SPLINE
SPL {X  -165.650, Y  +635.985, Z    +0.000, E1   -68.274, E3 +149186.290}
SPL {X  -165.650, Y  +656.072, Z    +0.000, E1   -68.403, E3 +149201.585}
SPL {X  -165.650, Y  +673.246, Z    +0.000, E1   -68.189, E3 +149217.340}
SPL {X  -164.760, Y  +692.647, Z    +0.000, E1   -68.400, E3 +149231.305}
SPL {X  -162.986, Y  +705.089, Z    +0.000, E1   -67.915, E3 +149245.517}
SPL {X  -160.378, Y  +716.957, Z    +0.000, E1   -67.874, E3 +149255.337}
SPL {X  -157.774, Y  +725.970, Z    +0.000, E1   -67.383, E3 +149266.685}
SPL {X  -154.751, Y  +734.593, Z    +0.000, E1   -66.864, E3 +149277.279}
SPL {X  -151.443, Y  +742.618, Z    +0.000, E1   -66.527, E3 +149286.274}
SPL {X  -148.198, Y  +749.508, Z    +0.000, E1   -66.065, E3 +149294.755}
SPL {X  -144.642, Y  +756.238, Z    +0.000, E1   -65.678, E3 +149302.621}
SPL {X  -140.398, Y  +763.411, Z    +0.000, E1   -64.853, E3 +149313.097}
SPL {X  -135.180, Y  +771.240, Z    +0.000, E1   -64.104, E3 +149323.147}
SPL {X  -125.028, Y  +784.164, Z    +0.000, E1   -66.760, E3 +149321.617}
SPL {X   -71.589, Y  +824.882, Z    +0.000, E1   -56.415, E3 +149448.682}
ENDSPLINE

SPLINE
SPL {X  -127.072, Y  +781.767, Z    +0.000, E1   -54.186, E3 +149611.654}
SPL {X  -150.680, Y  +744.314, Z    +0.000, E1   -44.608, E3 +149622.610}
SPL {X  -160.361, Y  +717.026, Z    +0.000, E1   -30.396, E3 +149611.464}
SPL {X  -163.361, Y  +702.946, Z    +0.000, E1   -22.646, E3 +149616.583}
SPL {X  -165.092, Y  +689.091, Z    +0.000, E1   -12.938, E3 +149616.153}
SPL {X  -165.629, Y  +678.122, Z    +0.000, E1    -4.178, E3 +149615.300}
SPL {X  -165.650, Y  +673.290, Z    +0.000, E1    +0.167, E3 +149614.256}
SPL {X  -165.650, Y  +669.039, Z    +0.000, E1    +7.218, E3 +149613.603}
SPL {X  -165.650, Y  +663.739, Z    +0.000, E1   +17.756, E3 +149613.294}
SPL {X  -165.650, Y  +659.573, Z    +0.000, E1   +26.182, E3 +149613.147}
SPL {X  -165.650, Y  +652.464, Z    +0.000, E1   +39.379, E3 +149612.188}
SPL {X  -165.650, Y  +634.871, Z    +0.000, E1   +61.762, E3 +149609.421}
SPL {X  -165.650, Y  +574.769, Z    +0.000, E1   +74.441, E3 +149622.069}
SPL {X  -165.650, Y  +420.321, Z    +0.000, E1   +71.570, E3 +149713.074}
ENDSPLINE

SPLINE
SPL {X  -165.650, Y  +437.633, Z    +0.000, E1   +68.421, E3 +149728.822}
ENDSPLINE

SPLINE
SPL {X  -164.513, Y  +359.128, Z    +0.000, E1   +73.170, E3 +149739.056}
SPL {X  -163.967, Y  +354.944, Z    +0.000, E1   +72.327, E3 +149750.409}
SPL {X  -163.372, Y  +351.124, Z    +0.000, E1   +71.295, E3 +149763.001}
SPL {X  -162.653, Y  +347.134, Z    +0.000, E1   +70.371, E3 +149774.237}
SPL {X  -161.430, Y  +341.349, Z    +0.000, E1   +69.492, E3 +149786.311}
SPL {X  -160.389, Y  +337.084, Z    +0.000, E1   +68.301, E3 +149799.398}
SPL {X  -159.245, Y  +332.881, Z    +0.000, E1   +67.496, E3 +149809.058}
SPL {X  -157.072, Y  +325.885, Z    +0.000, E1   +67.020, E3 +149818.407}
SPL {X  -154.432, Y  +318.577, Z    +0.000, E1   +66.843, E3 +149825.612}
SPL {X  -151.047, Y  +310.495, Z    +0.000, E1   +66.593, E3 +149834.024}
SPL {X  -146.639, Y  +301.448, Z    +0.000, E1   +65.839, E3 +149846.233}
SPL {X  -142.469, Y  +293.987, Z    +0.000, E1   +65.133, E3 +149856.282}
SPL {X  -139.022, Y  +288.429, Z    +0.000, E1   +64.807, E3 +149862.480}
SPL {X  -136.717, Y  +284.968, Z    +0.000, E1   +64.044, E3 +149869.073}
SPL {X  -133.061, Y  +279.835, Z    +0.000, E1   +64.204, E3 +149872.486}
SPL {X  -118.927, Y  +263.191, Z    +0.000, E1   +67.951, E3 +149868.499}
SPL {X   -76.819, Y  +231.739, Z    +0.000, E1   +54.834, E3 +150046.505}
ENDSPLINE

SPLINE
SPL {X  -140.879, Y  +291.363, Z    +0.000, E1   +48.273, E3 +150153.946}
SPL {X  -158.845, Y  +331.507, Z    +0.000, E1   +33.834, E3 +150163.281}
SPL {X  -164.164, Y  +356.358, Z    +0.000, E1   +18.707, E3 +150159.604}
SPL {X  -165.341, Y  +368.384, Z    +0.000, E1   +10.076, E3 +150160.348}
SPL {X  -165.648, Y  +377.641, Z    +0.000, E1    +2.653, E3 +150159.698}
SPL {X  -165.650, Y  +380.939, Z    +0.000, E1    -0.407, E3 +150158.509}
SPL {X  -165.650, Y  +385.900, Z    +0.000, E1    -8.711, E3 +150157.954}
SPL {X  -165.650, Y  +390.854, Z    +0.000, E1   -18.692, E3 +150157.129}
SPL {X  -165.650, Y  +395.801, Z    +0.000, E1   -28.236, E3 +150157.128}
SPL {X  -165.650, Y  +403.802, Z    +0.000, E1   -41.748, E3 +150156.949}
SPL {X  -165.650, Y  +418.088, Z    +0.000, E1   -59.974, E3 +150154.222}
SPL {X  -165.650, Y  +461.994, Z    +0.000, E1   -72.657, E3 +150162.360}
SPL {X  -165.650, Y  +492.072, Z    +0.000, E1   -73.925, E3 +150172.462}
SPL {X  -165.650, Y  +640.142, Z    +0.000, E1   -72.635, E3 +150251.338}
ENDSPLINE

SPLINE
SPL {X  -165.650, Y  +612.217, Z    +0.000, E1   -68.647, E3 +150267.263}
ENDSPLINE

SPLINE
SPL {X  -165.650, Y  +623.643, Z    +0.000, E1   -68.543, E3 +150277.360}
SPL {X  -165.650, Y  +635.985, Z    +0.000, E1   -68.274, E3 +150289.739}
SPL {X  -165.650, Y  +647.687, Z    +0.000, E1   -68.151, E3 +150300.238}
SPL {X  -165.650, Y  +665.917, Z    +0.000, E1   -68.414, E3 +150312.998}
SPL {X  -165.417, Y  +684.287, Z    +0.000, E1   -68.467, E3 +150327.295}
SPL {X  -164.655, Y  +693.631, Z    +0.000, E1   -68.130, E3 +150337.646}
SPL {X  -162.986, Y  +705.089, Z    +0.000, E1   -67.915, E3 +150348.965}
SPL {X  -159.812, Y  +719.091, Z    +0.000, E1   -67.711, E3 +150361.964}
SPL {X  -156.969, Y  +728.420, Z    +0.000, E1   -67.278, E3 +150372.746}
SPL {X  -154.751, Y  +734.593, Z    +0.000, E1   -66.864, E3 +150380.727}
SPL {X  -151.443, Y  +742.618, Z    +0.000, E1   -66.527, E3 +150389.722}
SPL {X  -148.198, Y  +749.508, Z    +0.000, E1   -66.065, E3 +150398.203}
SPL {X  -144.642, Y  +756.238, Z    +0.000, E1   -65.678, E3 +150406.070}
SPL {X  -140.398, Y  +763.411, Z    +0.000, E1   -64.853, E3 +150416.546}
SPL {X  -135.180, Y  +771.240, Z    +0.000, E1   -64.104, E3 +150426.595}
SPL {X  -125.028, Y  +784.164, Z    +0.000, E1   -66.760, E3 +150425.065}
SPL {X   -71.589, Y  +824.882, Z    +0.000, E1   -56.415, E3 +150552.130}
ENDSPLINE

SPLINE
SPL {X  -127.072, Y  +781.767, Z    +0.000, E1   -54.186, E3 +150715.102}
SPL {X  -150.680, Y  +744.314, Z    +0.000, E1   -44.608, E3 +150726.059}
SPL {X  -162.376, Y  +708.273, Z    +0.000, E1   -25.870, E3 +150718.182}
SPL {X  -165.092, Y  +689.091, Z    +0.000, E1   -12.938, E3 +150719.601}
SPL {X  -165.629, Y  +678.122, Z    +0.000, E1    -4.178, E3 +150718.748}
SPL {X  -165.650, Y  +673.539, Z    +0.000, E1    -0.057, E3 +150717.846}
SPL {X  -165.650, Y  +671.359, Z    +0.000, E1    +3.116, E3 +150717.203}
SPL {X  -165.650, Y  +667.465, Z    +0.000, E1   +10.413, E3 +150716.997}
SPL {X  -165.650, Y  +662.220, Z    +0.000, E1   +20.600, E3 +150716.689}
SPL {X  -165.650, Y  +652.464, Z    +0.000, E1   +39.379, E3 +150715.637}
SPL {X  -165.650, Y  +636.657, Z    +0.000, E1   +60.410, E3 +150712.925}
SPL {X  -165.650, Y  +613.310, Z    +0.000, E1   +72.038, E3 +150713.284}
SPL {X  -165.650, Y  +568.914, Z    +0.000, E1   +74.438, E3 +150727.869}
SPL {X  -165.650, Y  +420.321, Z    +0.000, E1   +71.570, E3 +150816.522}
ENDSPLINE

SPLINE
SPL {X  -165.650, Y  +437.633, Z    +0.000, E1   +68.421, E3 +150832.270}
ENDSPLINE

SPLINE
SPL {X  -164.513, Y  +359.128, Z    +0.000, E1   +73.170, E3 +150842.504}
SPL {X  -163.967, Y  +354.944, Z    +0.000, E1   +72.327, E3 +150853.857}
SPL {X  -163.372, Y  +351.124, Z    +0.000, E1   +71.295, E3 +150866.450}
SPL {X  -162.653, Y  +347.134, Z    +0.000, E1   +70.371, E3 +150877.685}
SPL {X  -161.451, Y  +341.438, Z    +0.000, E1   +69.889, E3 +150886.004}
SPL {X  -161.195, Y  +340.340, Z    +0.000, E1   +68.690, E3 +150897.225}
SPL {X  -159.328, Y  +333.173, Z    +0.000, E1   +67.752, E3 +150910.445}
SPL {X  -157.072, Y  +325.885, Z    +0.000, E1   +67.020, E3 +150921.855}
SPL {X  -154.432, Y  +318.577, Z    +0.000, E1   +66.843, E3 +150929.060}
SPL {X  -151.047, Y  +310.495, Z    +0.000, E1   +66.593, E3 +150937.472}
SPL {X  -146.639, Y  +301.448, Z    +0.000, E1   +65.839, E3 +150949.682}
SPL {X  -142.469, Y  +293.987, Z    +0.000, E1   +65.133, E3 +150959.730}
SPL {X  -139.022, Y  +288.429, Z    +0.000, E1   +64.807, E3 +150965.929}
SPL {X  -136.717, Y  +284.968, Z    +0.000, E1   +64.044, E3 +150972.521}
SPL {X  -133.061, Y  +279.835, Z    +0.000, E1   +64.204, E3 +150975.935}
SPL {X  -118.927, Y  +263.191, Z    +0.000, E1   +67.951, E3 +150971.947}
SPL {X   -76.819, Y  +231.739, Z    +0.000, E1   +54.834, E3 +151149.953}
ENDSPLINE

SPLINE
SPL {X  -140.879, Y  +291.363, Z    +0.000, E1   +48.273, E3 +151257.394}
SPL {X  -158.845, Y  +331.507, Z    +0.000, E1   +33.834, E3 +151266.729}
SPL {X  -164.164, Y  +356.358, Z    +0.000, E1   +18.707, E3 +151263.052}
SPL {X  -165.341, Y  +368.384, Z    +0.000, E1   +10.076, E3 +151263.796}
SPL {X  -165.648, Y  +377.641, Z    +0.000, E1    +2.653, E3 +151263.147}
SPL {X  -165.650, Y  +380.500, Z    +0.000, E1    -0.000, E3 +151262.177}
SPL {X  -165.650, Y  +381.694, Z    +0.000, E1    -1.679, E3 +151261.579}
SPL {X  -165.650, Y  +384.595, Z    +0.000, E1    -6.546, E3 +151261.441}
SPL {X  -165.650, Y  +389.276, Z    +0.000, E1   -15.245, E3 +151260.949}
SPL {X  -165.650, Y  +395.801, Z    +0.000, E1   -28.236, E3 +151260.576}
SPL {X  -165.650, Y  +403.802, Z    +0.000, E1   -41.748, E3 +151260.397}
SPL {X  -165.650, Y  +419.045, Z    +0.000, E1   -60.641, E3 +151257.718}
SPL {X  -165.650, Y  +466.630, Z    +0.000, E1   -73.161, E3 +151266.846}
SPL {X  -165.650, Y  +492.072, Z    +0.000, E1   -73.925, E3 +151275.910}
SPL {X  -165.650, Y  +637.039, Z    +0.000, E1   -73.842, E3 +151342.575}
ENDSPLINE

SPLINE
SPL {X  -165.650, Y  +617.598, Z    +0.000, E1   -69.273, E3 +151369.642}
ENDSPLINE

SPLINE
SPL {X  -165.650, Y  +623.643, Z    +0.000, E1   -68.543, E3 +151380.808}
SPL {X  -165.650, Y  +635.985, Z    +0.000, E1   -68.274, E3 +151393.187}
SPL {X  -165.650, Y  +656.072, Z    +0.000, E1   -68.403, E3 +151408.481}
SPL {X  -165.650, Y  +673.246, Z    +0.000, E1   -68.189, E3 +151424.236}
SPL {X  -164.760, Y  +692.647, Z    +0.000, E1   -68.400, E3 +151438.202}
SPL {X  -163.763, Y  +700.430, Z    +0.000, E1   -67.939, E3 +151448.225}
SPL {X  -161.478, Y  +712.444, Z    +0.000, E1   -67.895, E3 +151458.580}
SPL {X  -157.774, Y  +725.970, Z    +0.000, E1   -67.383, E3 +151473.581}
SPL {X  -153.458, Y  +737.875, Z    +0.000, E1   -66.902, E3 +151486.657}
SPL {X  -150.971, Y  +743.674, Z    +0.000, E1   -66.152, E3 +151496.314}
SPL {X  -146.969, Y  +751.920, Z    +0.000, E1   -66.066, E3 +151503.667}
SPL {X  -142.811, Y  +759.434, Z    +0.000, E1   -65.254, E3 +151514.516}
SPL {X  -139.420, Y  +764.954, Z    +0.000, E1   -64.577, E3 +151522.514}
SPL {X  -136.483, Y  +769.374, Z    +0.000, E1   -64.163, E3 +151528.169}
SPL {X  -133.523, Y  +773.539, Z    +0.000, E1   -63.962, E3 +151532.438}
SPL {X  -127.756, Y  +780.943, Z    +0.000, E1   -66.344, E3 +151528.032}
SPL {X  -118.855, Y  +790.884, Z    +0.000, E1   -67.633, E3 +151529.401}
SPL {X   -71.589, Y  +824.882, Z    +0.000, E1   -56.415, E3 +151655.578}
ENDSPLINE

SPLINE
SPL {X  -127.072, Y  +781.767, Z    +0.000, E1   -54.186, E3 +151818.550}
SPL {X  -150.680, Y  +744.314, Z    +0.000, E1   -44.608, E3 +151829.507}
SPL {X  -162.376, Y  +708.273, Z    +0.000, E1   -25.870, E3 +151821.630}
SPL {X  -165.092, Y  +689.091, Z    +0.000, E1   -12.938, E3 +151823.049}
SPL {X  -165.629, Y  +678.122, Z    +0.000, E1    -4.178, E3 +151822.196}
SPL {X  -165.650, Y  +673.539, Z    +0.000, E1    -0.057, E3 +151821.294}
SPL {X  -165.650, Y  +671.359, Z    +0.000, E1    +3.116, E3 +151820.651}
SPL {X  -165.650, Y  +667.465, Z    +0.000, E1   +10.413, E3 +151820.445}
SPL {X  -165.650, Y  +662.220, Z    +0.000, E1   +20.600, E3 +151820.137}
SPL {X  -165.650, Y  +652.464, Z    +0.000, E1   +39.379, E3 +151819.085}
SPL {X  -165.650, Y  +636.657, Z    +0.000, E1   +60.410, E3 +151816.373}
SPL {X  -165.650, Y  +613.310, Z    +0.000, E1   +72.038, E3 +151816.732}
SPL {X  -165.650, Y  +568.914, Z    +0.000, E1   +74.438, E3 +151831.317}
SPL {X  -165.650, Y  +420.321, Z    +0.000, E1   +71.570, E3 +151919.970}
ENDSPLINE

SPLINE
SPL {X  -165.650, Y  +437.633, Z    +0.000, E1   +68.421, E3 +151935.719}
ENDSPLINE

SPLINE
SPL {X  -164.513, Y  +359.128, Z    +0.000, E1   +73.170, E3 +151945.952}
SPL {X  -163.967, Y  +354.944, Z    +0.000, E1   +72.327, E3 +151957.306}
SPL {X  -163.372, Y  +351.124, Z    +0.000, E1   +71.295, E3 +151969.898}
SPL {X  -162.653, Y  +347.134, Z    +0.000, E1   +70.371, E3 +151981.133}
SPL {X  -161.451, Y  +341.438, Z    +0.000, E1   +69.889, E3 +151989.452}
SPL {X  -161.195, Y  +340.340, Z    +0.000, E1   +68.690, E3 +152000.673}
SPL {X  -159.328, Y  +333.173, Z    +0.000, E1   +67.752, E3 +152013.894}
SPL {X  -157.072, Y  +325.885, Z    +0.000, E1   +67.020, E3 +152025.304}
SPL {X  -154.432, Y  +318.577, Z    +0.000, E1   +66.843, E3 +152032.509}
SPL {X  -151.047, Y  +310.495, Z    +0.000, E1   +66.593, E3 +152040.921}
SPL {X  -146.639, Y  +301.448, Z    +0.000, E1   +65.839, E3 +152053.130}
SPL {X  -142.469, Y  +293.987, Z    +0.000, E1   +65.133, E3 +152063.178}
SPL {X  -139.022, Y  +288.429, Z    +0.000, E1   +64.807, E3 +152069.377}
SPL {X  -136.717, Y  +284.968, Z    +0.000, E1   +64.044, E3 +152075.969}
SPL {X  -133.061, Y  +279.835, Z    +0.000, E1   +64.204, E3 +152079.383}
SPL {X  -118.927, Y  +263.191, Z    +0.000, E1   +67.951, E3 +152075.395}
SPL {X   -76.819, Y  +231.739, Z    +0.000, E1   +54.834, E3 +152253.402}
ENDSPLINE

SPLINE
SPL {X  -140.879, Y  +291.363, Z    +0.000, E1   +48.273, E3 +152360.843}
SPL {X  -158.845, Y  +331.507, Z    +0.000, E1   +33.834, E3 +152370.178}
SPL {X  -164.164, Y  +356.358, Z    +0.000, E1   +18.707, E3 +152366.500}
SPL {X  -165.341, Y  +368.384, Z    +0.000, E1   +10.076, E3 +152367.244}
SPL {X  -165.648, Y  +377.641, Z    +0.000, E1    +2.653, E3 +152366.595}
SPL {X  -165.650, Y  +380.500, Z    +0.000, E1    -0.000, E3 +152365.626}
SPL {X  -165.650, Y  +381.694, Z    +0.000, E1    -1.679, E3 +152365.027}
SPL {X  -165.650, Y  +384.595, Z    +0.000, E1    -6.546, E3 +152364.889}
SPL {X  -165.650, Y  +389.276, Z    +0.000, E1   -15.245, E3 +152364.397}
SPL {X  -165.650, Y  +395.801, Z    +0.000, E1   -28.236, E3 +152364.025}
SPL {X  -165.650, Y  +403.802, Z    +0.000, E1   -41.748, E3 +152363.846}
SPL {X  -165.650, Y  +419.045, Z    +0.000, E1   -60.641, E3 +152361.167}
SPL {X  -165.650, Y  +474.102, Z    +0.000, E1   -73.446, E3 +152372.950}
SPL {X  -165.650, Y  +640.142, Z    +0.000, E1   -72.635, E3 +152458.235}
ENDSPLINE

SPLINE
SPL {X  -165.650, Y  +619.423, Z    +0.000, E1   -68.618, E3 +152480.432}
ENDSPLINE

SPLINE
SPL {X  -165.650, Y  +635.985, Z    +0.000, E1   -68.274, E3 +152496.635}
SPL {X  -165.650, Y  +647.687, Z    +0.000, E1   -68.151, E3 +152507.135}
SPL {X  -165.650, Y  +665.917, Z    +0.000, E1   -68.414, E3 +152519.894}
SPL {X  -165.417, Y  +684.287, Z    +0.000, E1   -68.467, E3 +152534.192}
SPL {X  -164.268, Y  +696.853, Z    +0.000, E1   -68.071, E3 +152547.821}
SPL {X  -161.478, Y  +712.444, Z    +0.000, E1   -67.895, E3 +152562.028}
SPL {X  -157.774, Y  +725.970, Z    +0.000, E1   -67.383, E3 +152577.029}
SPL {X  -154.751, Y  +734.593, Z    +0.000, E1   -66.864, E3 +152587.624}
SPL {X  -151.443, Y  +742.618, Z    +0.000, E1   -66.527, E3 +152596.619}
SPL {X  -146.969, Y  +751.920, Z    +0.000, E1   -66.066, E3 +152607.115}
SPL {X  -142.811, Y  +759.434, Z    +0.000, E1   -65.254, E3 +152617.964}
SPL {X  -139.420, Y  +764.954, Z    +0.000, E1   -64.577, E3 +152625.963}
SPL {X  -136.483, Y  +769.374, Z    +0.000, E1   -64.163, E3 +152631.618}
SPL {X  -133.523, Y  +773.539, Z    +0.000, E1   -63.962, E3 +152635.886}
SPL {X  -125.028, Y  +784.164, Z    +0.000, E1   -66.760, E3 +152631.962}
SPL {X   -71.589, Y  +824.882, Z    +0.000, E1   -56.415, E3 +152759.027}
ENDSPLINE

SPLINE
SPL {X  -127.072, Y  +781.767, Z    +0.000, E1   -54.186, E3 +152921.999}
SPL {X  -150.680, Y  +744.314, Z    +0.000, E1   -44.608, E3 +152932.955}
SPL {X  -162.376, Y  +708.273, Z    +0.000, E1   -25.870, E3 +152925.079}
SPL {X  -165.092, Y  +689.091, Z    +0.000, E1   -12.938, E3 +152926.498}
SPL {X  -165.629, Y  +678.122, Z    +0.000, E1    -4.178, E3 +152925.645}
SPL {X  -165.650, Y  +673.539, Z    +0.000, E1    -0.057, E3 +152924.742}
SPL {X  -165.650, Y  +671.359, Z    +0.000, E1    +3.116, E3 +152924.099}
SPL {X  -165.650, Y  +665.277, Z    +0.000, E1   +14.409, E3 +152923.744}
SPL {X  -165.650, Y  +659.573, Z    +0.000, E1   +26.182, E3 +152923.492}
SPL {X  -165.650, Y  +652.464, Z    +0.000, E1   +39.379, E3 +152922.533}
SPL {X  -165.650, Y  +634.871, Z    +0.000, E1   +61.762, E3 +152919.766}
SPL {X  -165.650, Y  +574.769, Z    +0.000, E1   +74.441, E3 +152932.414}
SPL {X  -165.650, Y  +420.321, Z    +0.000, E1   +71.570, E3 +153023.419}
ENDSPLINE

SPLINE
SPL {X  -165.650, Y  +437.633, Z    +0.000, E1   +68.421, E3 +153039.167}
ENDSPLINE

SPLINE
SPL {X  -164.513, Y  +359.128, Z    +0.000, E1   +73.170, E3 +153049.401}
SPL {X  -163.967, Y  +354.944, Z    +0.000, E1   +72.327, E3 +153060.754}
SPL {X  -163.372, Y  +351.124, Z    +0.000, E1   +71.295, E3 +153073.346}
SPL {X  -162.653, Y  +347.134, Z    +0.000, E1   +70.371, E3 +153084.581}
SPL {X  -161.430, Y  +341.349, Z    +0.000, E1   +69.492, E3 +153096.656}
SPL {X  -160.389, Y  +337.084, Z    +0.000, E1   +68.301, E3 +153109.743}
SPL {X  -158.795, Y  +331.340, Z    +0.000, E1   +67.291, E3 +153122.429}
SPL {X  -155.058, Y  +320.218, Z    +0.000, E1   +66.982, E3 +153133.735}
SPL {X  -151.047, Y  +310.495, Z    +0.000, E1   +66.593, E3 +153144.369}
SPL {X  -148.187, Y  +304.469, Z    +0.000, E1   +66.029, E3 +153152.748}
SPL {X  -145.703, Y  +299.692, Z    +0.000, E1   +65.663, E3 +153158.914}
SPL {X  -142.469, Y  +293.987, Z    +0.000, E1   +65.133, E3 +153166.627}
SPL {X  -139.022, Y  +288.429, Z    +0.000, E1   +64.807, E3 +153172.825}
SPL {X  -136.717, Y  +284.968, Z    +0.000, E1   +64.044, E3 +153179.418}
SPL {X  -133.061, Y  +279.835, Z    +0.000, E1   +64.204, E3 +153182.831}
SPL {X  -118.927, Y  +263.191, Z    +0.000, E1   +67.951, E3 +153178.844}
SPL {X   -76.819, Y  +231.739, Z    +0.000, E1   +54.834, E3 +153356.850}
ENDSPLINE

SPLINE
SPL {X  -140.879, Y  +291.363, Z    +0.000, E1   +48.273, E3 +153464.291}
SPL {X  -158.845, Y  +331.507, Z    +0.000, E1   +33.834, E3 +153473.626}
SPL {X  -164.164, Y  +356.358, Z    +0.000, E1   +18.707, E3 +153469.948}
SPL {X  -165.519, Y  +371.910, Z    +0.000, E1    +7.409, E3 +153470.357}
SPL {X  -165.650, Y  +380.329, Z    +0.000, E1    +0.239, E3 +153469.203}
SPL {X  -165.650, Y  +381.694, Z    +0.000, E1    -1.679, E3 +153468.475}
SPL {X  -165.650, Y  +384.595, Z    +0.000, E1    -6.546, E3 +153468.338}
SPL {X  -165.650, Y  +389.276, Z    +0.000, E1   -15.245, E3 +153467.846}
SPL {X  -165.650, Y  +395.801, Z    +0.000, E1   -28.236, E3 +153467.473}
SPL {X  -165.650, Y  +403.802, Z    +0.000, E1   -41.748, E3 +153467.294}
SPL {X  -165.650, Y  +418.088, Z    +0.000, E1   -59.974, E3 +153464.567}
SPL {X  -165.650, Y  +461.994, Z    +0.000, E1   -72.657, E3 +153472.704}
SPL {X  -165.650, Y  +492.072, Z    +0.000, E1   -73.925, E3 +153482.807}
SPL {X  -165.650, Y  +640.142, Z    +0.000, E1   -72.635, E3 +153561.683}
ENDSPLINE

SPLINE
SPL {X  -165.650, Y  +619.423, Z    +0.000, E1   -68.618, E3 +153583.880}
ENDSPLINE

SPLINE
SPL {X  -165.650, Y  +635.985, Z    +0.000, E1   -68.274, E3 +153600.083}
SPL {X  -165.650, Y  +647.687, Z    +0.000, E1   -68.151, E3 +153610.583}
SPL {X  -165.650, Y  +662.755, Z    +0.000, E1   -68.565, E3 +153619.250}
SPL {X  -165.650, Y  +673.246, Z    +0.000, E1   -68.189, E3 +153631.133}
SPL {X  -164.760, Y  +692.647, Z    +0.000, E1   -68.400, E3 +153645.098}
SPL {X  -163.763, Y  +700.430, Z    +0.000, E1   -67.939, E3 +153655.121}
SPL {X  -162.443, Y  +707.938, Z    +0.000, E1   -67.853, E3 +153662.003}
SPL {X  -159.812, Y  +719.091, Z    +0.000, E1   -67.711, E3 +153672.309}
SPL {X  -156.969, Y  +728.420, Z    +0.000, E1   -67.278, E3 +153683.091}
SPL {X  -154.751, Y  +734.593, Z    +0.000, E1   -66.864, E3 +153691.072}
SPL {X  -151.443, Y  +742.618, Z    +0.000, E1   -66.527, E3 +153700.067}
SPL {X  -148.198, Y  +749.508, Z    +0.000, E1   -66.065, E3 +153708.548}
SPL {X  -144.642, Y  +756.238, Z    +0.000, E1   -65.678, E3 +153716.414}
SPL {X  -140.398, Y  +763.411, Z    +0.000, E1   -64.853, E3 +153726.891}
SPL {X  -135.180, Y  +771.240, Z    +0.000, E1   -64.104, E3 +153736.940}
SPL {X  -125.028, Y  +784.164, Z    +0.000, E1   -66.760, E3 +153735.410}
SPL {X   -71.589, Y  +824.882, Z    +0.000, E1   -56.415, E3 +153862.475}
ENDSPLINE

SPLINE
SPL {X  -127.072, Y  +781.767, Z    +0.000, E1   -54.186, E3 +154025.447}
SPL {X  -150.680, Y  +744.314, Z    +0.000, E1   -44.608, E3 +154036.403}
SPL {X  -162.376, Y  +708.273, Z    +0.000, E1   -25.870, E3 +154028.527}
SPL {X  -165.092, Y  +689.091, Z    +0.000, E1   -12.938, E3 +154029.946}
SPL {X  -165.629, Y  +678.122, Z    +0.000, E1    -4.178, E3 +154029.093}
SPL {X  -165.650, Y  +673.290, Z    +0.000, E1    +0.167, E3 +154028.049}
SPL {X  -165.650, Y  +669.039, Z    +0.000, E1    +7.218, E3 +154027.396}
SPL {X  -165.650, Y  +662.220, Z    +0.000, E1   +20.600, E3 +154027.034}
SPL {X  -165.650, Y  +652.464, Z    +0.000, E1   +39.379, E3 +154025.981}
SPL {X  -165.650, Y  +634.871, Z    +0.000, E1   +61.762, E3 +154023.214}
SPL {X  -165.650, Y  +574.769, Z    +0.000, E1   +74.441, E3 +154035.862}
SPL {X  -165.650, Y  +420.321, Z    +0.000, E1   +71.570, E3 +154126.867}
ENDSPLINE

SPLINE
SPL {X  -165.650, Y  +437.633, Z    +0.000, E1   +68.421, E3 +154142.615}
ENDSPLINE

SPLINE
SPL {X  -164.513, Y  +359.128, Z    +0.000, E1   +73.170, E3 +154152.849}
SPL {X  -163.967, Y  +354.944, Z    +0.000, E1   +72.327, E3 +154164.202}
SPL {X  -163.372, Y  +351.124, Z    +0.000, E1   +71.295, E3 +154176.794}
SPL {X  -162.653, Y  +347.134, Z    +0.000, E1   +70.371, E3 +154188.030}
SPL {X  -161.430, Y  +341.349, Z    +0.000, E1   +69.492, E3 +154200.104}
SPL {X  -160.389, Y  +337.084, Z    +0.000, E1   +68.301, E3 +154213.191}
SPL {X  -159.245, Y  +332.881, Z    +0.000, E1   +67.496, E3 +154222.851}
SPL {X  -157.072, Y  +325.885, Z    +0.000, E1   +67.020, E3 +154232.200}
SPL {X  -154.432, Y  +318.577, Z    +0.000, E1   +66.843, E3 +154239.405}
SPL {X  -151.047, Y  +310.495, Z    +0.000, E1   +66.593, E3 +154247.817}
SPL {X  -148.187, Y  +304.469, Z    +0.000, E1   +66.029, E3 +154256.196}
SPL {X  -145.703, Y  +299.692, Z    +0.000, E1   +65.663, E3 +154262.362}
SPL {X  -142.469, Y  +293.987, Z    +0.000, E1   +65.133, E3 +154270.075}
SPL {X  -139.022, Y  +288.429, Z    +0.000, E1   +64.807, E3 +154276.274}
SPL {X  -136.717, Y  +284.968, Z    +0.000, E1   +64.044, E3 +154282.866}
SPL {X  -133.061, Y  +279.835, Z    +0.000, E1   +64.204, E3 +154286.280}
SPL {X  -118.927, Y  +263.191, Z    +0.000, E1   +67.951, E3 +154282.292}
SPL {X   -76.819, Y  +231.739, Z    +0.000, E1   +54.834, E3 +154460.298}
ENDSPLINE

SPLINE
SPL {X  -140.879, Y  +291.363, Z    +0.000, E1   +48.273, E3 +154567.739}
SPL {X  -155.054, Y  +320.205, Z    +0.000, E1   +39.591, E3 +154580.191}
SPL {X  -160.978, Y  +339.437, Z    +0.000, E1   +29.257, E3 +154574.820}
SPL {X  -164.164, Y  +356.358, Z    +0.000, E1   +18.707, E3 +154573.397}
SPL {X  -165.519, Y  +371.910, Z    +0.000, E1    +7.409, E3 +154573.806}
SPL {X  -165.650, Y  +380.329, Z    +0.000, E1    +0.239, E3 +154572.652}
SPL {X  -165.650, Y  +381.694, Z    +0.000, E1    -1.679, E3 +154571.924}
SPL {X  -165.650, Y  +384.595, Z    +0.000, E1    -6.546, E3 +154571.786}
SPL {X  -165.650, Y  +389.276, Z    +0.000, E1   -15.245, E3 +154571.294}
SPL {X  -165.650, Y  +395.801, Z    +0.000, E1   -28.236, E3 +154570.921}
SPL {X  -165.650, Y  +403.802, Z    +0.000, E1   -41.748, E3 +154570.742}
SPL {X  -165.650, Y  +419.045, Z    +0.000, E1   -60.641, E3 +154568.063}
SPL {X  -165.650, Y  +474.102, Z    +0.000, E1   -73.446, E3 +154579.846}
SPL {X  -165.650, Y  +640.142, Z    +0.000, E1   -72.635, E3 +154665.131}
ENDSPLINE

SPLINE
SPL {X  -165.650, Y  +612.217, Z    +0.000, E1   -68.647, E3 +154681.056}
ENDSPLINE

SPLINE
SPL {X  -165.650, Y  +623.643, Z    +0.000, E1   -68.543, E3 +154691.153}
SPL {X  -165.650, Y  +635.985, Z    +0.000, E1   -68.274, E3 +154703.532}
SPL {X  -165.650, Y  +647.687, Z    +0.000, E1   -68.151, E3 +154714.031}
SPL {X  -165.650, Y  +665.917, Z    +0.000, E1   -68.414, E3 +154726.791}
SPL {X  -165.417, Y  +684.287, Z    +0.000, E1   -68.467, E3 +154741.088}
SPL {X  -164.268, Y  +696.853, Z    +0.000, E1   -68.071, E3 +154754.717}
SPL {X  -162.443, Y  +707.938, Z    +0.000, E1   -67.853, E3 +154765.452}
SPL {X  -159.812, Y  +719.091, Z    +0.000, E1   -67.711, E3 +154775.757}
SPL {X  -156.969, Y  +728.420, Z    +0.000, E1   -67.278, E3 +154786.539}
SPL {X  -154.751, Y  +734.593, Z    +0.000, E1   -66.864, E3 +154794.520}
SPL {X  -151.443, Y  +742.618, Z    +0.000, E1   -66.527, E3 +154803.515}
SPL {X  -146.969, Y  +751.920, Z    +0.000, E1   -66.066, E3 +154814.012}
SPL {X  -142.811, Y  +759.434, Z    +0.000, E1   -65.254, E3 +154824.860}
SPL {X  -139.420, Y  +764.954, Z    +0.000, E1   -64.577, E3 +154832.859}
SPL {X  -136.483, Y  +769.374, Z    +0.000, E1   -64.163, E3 +154838.514}
SPL {X  -133.523, Y  +773.539, Z    +0.000, E1   -63.962, E3 +154842.783}
SPL {X  -125.028, Y  +784.164, Z    +0.000, E1   -66.760, E3 +154838.858}
SPL {X   -71.589, Y  +824.882, Z    +0.000, E1   -56.415, E3 +154965.923}
ENDSPLINE

SPLINE
SPL {X  -127.072, Y  +781.767, Z    +0.000, E1   -54.186, E3 +155128.895}
SPL {X  -150.680, Y  +744.314, Z    +0.000, E1   -44.608, E3 +155139.852}
SPL {X  -162.376, Y  +708.273, Z    +0.000, E1   -25.870, E3 +155131.975}
SPL {X  -165.092, Y  +689.091, Z    +0.000, E1   -12.938, E3 +155133.394}
SPL {X  -165.569, Y  +680.695, Z    +0.000, E1    -6.245, E3 +155132.079}
SPL {X  -165.650, Y  +673.489, Z    +0.000, E1    -0.162, E3 +155131.584}
SPL {X  -165.650, Y  +669.039, Z    +0.000, E1    +7.218, E3 +155130.845}
SPL {X  -165.650, Y  +662.220, Z    +0.000, E1   +20.600, E3 +155130.482}
SPL {X  -165.650, Y  +652.464, Z    +0.000, E1   +39.379, E3 +155129.430}
SPL {X  -165.650, Y  +636.657, Z    +0.000, E1   +60.410, E3 +155126.718}
SPL {X  -165.650, Y  +613.310, Z    +0.000, E1   +72.038, E3 +155127.077}
SPL {X  -165.650, Y  +568.914, Z    +0.000, E1   +74.438, E3 +155141.662}
SPL {X  -165.650, Y  +420.321, Z    +0.000, E1   +71.570, E3 +155230.315}
ENDSPLINE

SPLINE
SPL {X  -165.650, Y  +437.633, Z    +0.000, E1   +68.421, E3 +155246.064}
ENDSPLINE

SPLINE
SPL {X  -164.513, Y  +359.128, Z    +0.000, E1   +73.170, E3 +155256.297}
SPL {X  -163.967, Y  +354.944, Z    +0.000, E1   +72.327, E3 +155267.650}
SPL {X  -163.571, Y  +352.336, Z    +0.000, E1   +71.524, E3 +155277.068}
SPL {X  -162.836, Y  +348.099, Z    +0.000, E1   +70.646, E3 +155288.542}
SPL {X  -161.451, Y  +341.438, Z    +0.000, E1   +69.889, E3 +155299.797}
SPL {X  -161.444, Y  +341.410, Z    +0.000, E1   +69.001, E3 +155307.384}
SPL {X  -160.389, Y  +337.084, Z    +0.000, E1   +68.301, E3 +155316.640}
SPL {X  -159.245, Y  +332.881, Z    +0.000, E1   +67.496, E3 +155326.299}
SPL {X  -157.072, Y  +325.885, Z    +0.000, E1   +67.020, E3 +155335.648}
SPL {X  -153.570, Y  +316.402, Z    +0.000, E1   +66.799, E3 +155345.010}
SPL {X  -150.243, Y  +308.737, Z    +0.000, E1   +66.492, E3 +155353.252}
SPL {X  -146.639, Y  +301.448, Z    +0.000, E1   +65.839, E3 +155363.475}
SPL {X  -142.469, Y  +293.987, Z    +0.000, E1   +65.133, E3 +155373.523}
SPL {X  -139.022, Y  +288.429, Z    +0.000, E1   +64.807, E3 +155379.722}
SPL {X  -136.717, Y  +284.968, Z    +0.000, E1   +64.044, E3 +155386.314}
SPL {X  -133.061, Y  +279.835, Z    +0.000, E1   +64.204, E3 +155389.728}
SPL {X  -118.927, Y  +263.191, Z    +0.000, E1   +67.951, E3 +155385.740}
SPL {X   -76.819, Y  +231.739, Z    +0.000, E1   +54.834, E3 +155563.746}
ENDSPLINE

SPLINE
SPL {X  -140.879, Y  +291.363, Z    +0.000, E1   +48.273, E3 +155671.188}
SPL {X  -158.845, Y  +331.507, Z    +0.000, E1   +33.834, E3 +155680.522}
SPL {X  -164.164, Y  +356.358, Z    +0.000, E1   +18.707, E3 +155676.845}
SPL {X  -165.341, Y  +368.384, Z    +0.000, E1   +10.076, E3 +155677.589}
SPL {X  -165.648, Y  +377.641, Z    +0.000, E1    +2.653, E3 +155676.940}
SPL {X  -165.650, Y  +380.939, Z    +0.000, E1    -0.407, E3 +155675.750}
SPL {X  -165.650, Y  +385.900, Z    +0.000, E1    -8.711, E3 +155675.195}
SPL {X  -165.650, Y  +390.854, Z    +0.000, E1   -18.692, E3 +155674.371}
SPL {X  -165.650, Y  +395.801, Z    +0.000, E1   -28.236, E3 +155674.370}
SPL {X  -165.650, Y  +403.802, Z    +0.000, E1   -41.748, E3 +155674.190}
SPL {X  -165.650, Y  +418.088, Z    +0.000, E1   -59.974, E3 +155671.463}
SPL {X  -165.650, Y  +461.994, Z    +0.000, E1   -72.657, E3 +155679.601}
SPL {X  -165.650, Y  +492.072, Z    +0.000, E1   -73.925, E3 +155689.703}
SPL {X  -165.650, Y  +640.142, Z    +0.000, E1   -72.635, E3 +155768.579}
ENDSPLINE

SPLINE
SPL {X  -165.650, Y  +619.423, Z    +0.000, E1   -68.618, E3 +155790.777}
ENDSPLINE

SPLINE
SPL {X  -165.650, Y  +635.985, Z    +0.000, E1   -68.274, E3 +155806.980}
SPL {X  -165.650, Y  +656.072, Z    +0.000, E1   -68.403, E3 +155822.274}
SPL {X  -165.650, Y  +673.246, Z    +0.000, E1   -68.189, E3 +155838.030}
SPL {X  -164.760, Y  +692.647, Z    +0.000, E1   -68.400, E3 +155851.995}
SPL {X  -162.986, Y  +705.089, Z    +0.000, E1   -67.915, E3 +155866.207}
SPL {X  -159.812, Y  +719.091, Z    +0.000, E1   -67.711, E3 +155879.206}
SPL {X  -156.969, Y  +728.420, Z    +0.000, E1   -67.278, E3 +155889.988}
SPL {X  -154.751, Y  +734.593, Z    +0.000, E1   -66.864, E3 +155897.969}
SPL {X  -151.443, Y  +742.618, Z    +0.000, E1   -66.527, E3 +155906.964}
SPL {X  -146.969, Y  +751.920, Z    +0.000, E1   -66.066, E3 +155917.460}
SPL {X  -142.811, Y  +759.434, Z    +0.000, E1   -65.254, E3 +155928.309}
SPL {X  -139.420, Y  +764.954, Z    +0.000, E1   -64.577, E3 +155936.307}
SPL {X  -136.483, Y  +769.374, Z    +0.000, E1   -64.163, E3 +155941.962}
SPL {X  -133.523, Y  +773.539, Z    +0.000, E1   -63.962, E3 +155946.231}
SPL {X  -125.028, Y  +784.164, Z    +0.000, E1   -66.760, E3 +155942.306}
SPL {X   -71.589, Y  +824.882, Z    +0.000, E1   -56.415, E3 +156069.371}
ENDSPLINE

SPLINE
SPL {X  -127.072, Y  +781.767, Z    +0.000, E1   -54.186, E3 +156232.344}
SPL {X  -150.680, Y  +744.314, Z    +0.000, E1   -44.608, E3 +156243.300}
SPL {X  -162.376, Y  +708.273, Z    +0.000, E1   -25.870, E3 +156235.424}
SPL {X  -165.092, Y  +689.091, Z    +0.000, E1   -12.938, E3 +156236.842}
SPL {X  -165.569, Y  +680.695, Z    +0.000, E1    -6.245, E3 +156235.528}
SPL {X  -165.650, Y  +673.489, Z    +0.000, E1    -0.162, E3 +156235.032}
SPL {X  -165.650, Y  +669.039, Z    +0.000, E1    +7.218, E3 +156234.293}
SPL {X  -165.650, Y  +663.739, Z    +0.000, E1   +17.756, E3 +156233.984}
SPL {X  -165.650, Y  +659.573, Z    +0.000, E1   +26.182, E3 +156233.837}
SPL {X  -165.650, Y  +652.464, Z    +0.000, E1   +39.379, E3 +156232.878}
SPL {X  -165.650, Y  +634.871, Z    +0.000, E1   +61.762, E3 +156230.110}
SPL {X  -165.650, Y  +574.769, Z    +0.000, E1   +74.441, E3 +156242.759}
SPL {X  -165.650, Y  +420.321, Z    +0.000, E1   +71.570, E3 +156333.763}
ENDSPLINE

SPLINE
SPL {X  -165.650, Y  +437.633, Z    +0.000, E1   +68.421, E3 +156349.512}
ENDSPLINE

SPLINE
SPL {X  -164.513, Y  +359.128, Z    +0.000, E1   +73.170, E3 +156359.745}
SPL {X  -163.967, Y  +354.944, Z    +0.000, E1   +72.327, E3 +156371.099}
SPL {X  -163.571, Y  +352.336, Z    +0.000, E1   +71.524, E3 +156380.517}
SPL {X  -162.836, Y  +348.099, Z    +0.000, E1   +70.646, E3 +156391.990}
SPL {X  -161.451, Y  +341.438, Z    +0.000, E1   +69.889, E3 +156403.245}
SPL {X  -161.195, Y  +340.340, Z    +0.000, E1   +68.690, E3 +156414.466}
SPL {X  -159.328, Y  +333.173, Z    +0.000, E1   +67.752, E3 +156427.687}
SPL {X  -157.072, Y  +325.885, Z    +0.000, E1   +67.020, E3 +156439.097}
SPL {X  -154.432, Y  +318.577, Z    +0.000, E1   +66.843, E3 +156446.302}
SPL {X  -151.047, Y  +310.495, Z    +0.000, E1   +66.593, E3 +156454.714}
SPL {X  -146.639, Y  +301.448, Z    +0.000, E1   +65.839, E3 +156466.923}
SPL {X  -142.469, Y  +293.987, Z    +0.000, E1   +65.133, E3 +156476.972}
SPL {X  -139.022, Y  +288.429, Z    +0.000, E1   +64.807, E3 +156483.170}
SPL {X  -136.717, Y  +284.968, Z    +0.000, E1   +64.044, E3 +156489.763}
SPL {X  -133.061, Y  +279.835, Z    +0.000, E1   +64.204, E3 +156493.176}
SPL {X  -118.927, Y  +263.191, Z    +0.000, E1   +67.951, E3 +156489.189}
SPL {X   -76.819, Y  +231.739, Z    +0.000, E1   +54.834, E3 +156667.195}
ENDSPLINE

SPLINE
SPL {X  -140.879, Y  +291.363, Z    +0.000, E1   +48.273, E3 +156774.636}
SPL {X  -158.845, Y  +331.507, Z    +0.000, E1   +33.834, E3 +156783.971}
SPL {X  -164.164, Y  +356.358, Z    +0.000, E1   +18.707, E3 +156780.293}
SPL {X  -165.341, Y  +368.384, Z    +0.000, E1   +10.076, E3 +156781.037}
SPL {X  -165.648, Y  +377.641, Z    +0.000, E1    +2.653, E3 +156780.388}
SPL {X  -165.650, Y  +380.500, Z    +0.000, E1    -0.000, E3 +156779.419}
SPL {X  -165.650, Y  +381.694, Z    +0.000, E1    -1.679, E3 +156778.820}
SPL {X  -165.650, Y  +384.595, Z    +0.000, E1    -6.546, E3 +156778.682}
SPL {X  -165.650, Y  +389.276, Z    +0.000, E1   -15.245, E3 +156778.191}
SPL {X  -165.650, Y  +395.801, Z    +0.000, E1   -28.236, E3 +156777.818}
SPL {X  -165.650, Y  +403.802, Z    +0.000, E1   -41.748, E3 +156777.639}
SPL {X  -165.650, Y  +419.045, Z    +0.000, E1   -60.641, E3 +156774.960}
SPL {X  -165.650, Y  +474.102, Z    +0.000, E1   -73.446, E3 +156786.743}
SPL {X  -165.650, Y  +640.142, Z    +0.000, E1   -72.635, E3 +156872.028}
ENDSPLINE

SPLINE
SPL {X  -165.650, Y  +612.217, Z    +0.000, E1   -68.647, E3 +156887.953}
ENDSPLINE

SPLINE
SPL {X  -165.650, Y  +623.643, Z    +0.000, E1   -68.543, E3 +156898.050}
SPL {X  -165.650, Y  +635.985, Z    +0.000, E1   -68.274, E3 +156910.428}
SPL {X  -165.650, Y  +656.072, Z    +0.000, E1   -68.403, E3 +156925.723}
SPL {X  -165.650, Y  +673.246, Z    +0.000, E1   -68.189, E3 +156941.478}
SPL {X  -164.760, Y  +692.647, Z    +0.000, E1   -68.400, E3 +156955.443}
SPL {X  -162.986, Y  +705.089, Z    +0.000, E1   -67.915, E3 +156969.655}
SPL {X  -159.812, Y  +719.091, Z    +0.000, E1   -67.711, E3 +156982.654}
SPL {X  -156.969, Y  +728.420, Z    +0.000, E1   -67.278, E3 +156993.436}
SPL {X  -154.751, Y  +734.593, Z    +0.000, E1   -66.864, E3 +157001.417}
SPL {X  -151.443, Y  +742.618, Z    +0.000, E1   -66.527, E3 +157010.412}
SPL {X  -146.969, Y  +751.920, Z    +0.000, E1   -66.066, E3 +157020.909}
SPL {X  -142.811, Y  +759.434, Z    +0.000, E1   -65.254, E3 +157031.757}
SPL {X  -139.420, Y  +764.954, Z    +0.000, E1   -64.577, E3 +157039.756}
SPL {X  -136.483, Y  +769.374, Z    +0.000, E1   -64.163, E3 +157045.411}
SPL {X  -133.523, Y  +773.539, Z    +0.000, E1   -63.962, E3 +157049.679}
SPL {X  -125.028, Y  +784.164, Z    +0.000, E1   -66.760, E3 +157045.755}
SPL {X   -71.589, Y  +824.882, Z    +0.000, E1   -56.415, E3 +157172.820}
ENDSPLINE

SPLINE
SPL {X  -127.072, Y  +781.767, Z    +0.000, E1   -54.186, E3 +157335.792}
SPL {X  -150.680, Y  +744.314, Z    +0.000, E1   -44.608, E3 +157346.748}
SPL {X  -162.376, Y  +708.273, Z    +0.000, E1   -25.870, E3 +157338.872}
SPL {X  -165.092, Y  +689.091, Z    +0.000, E1   -12.938, E3 +157340.291}
SPL {X  -165.569, Y  +680.695, Z    +0.000, E1    -6.245, E3 +157338.976}
SPL {X  -165.650, Y  +673.489, Z    +0.000, E1    -0.162, E3 +157338.480}
SPL {X  -165.650, Y  +669.039, Z    +0.000, E1    +7.218, E3 +157337.741}
SPL {X  -165.650, Y  +663.739, Z    +0.000, E1   +17.756, E3 +157337.432}
SPL {X  -165.650, Y  +656.188, Z    +0.000, E1   +32.567, E3 +157336.714}
SPL {X  -165.650, Y  +648.712, Z    +0.000, E1   +45.195, E3 +157336.336}
SPL {X  -165.650, Y  +636.657, Z    +0.000, E1   +60.410, E3 +157333.614}
SPL {X  -165.650, Y  +613.310, Z    +0.000, E1   +72.038, E3 +157333.974}
SPL {X  -165.650, Y  +568.914, Z    +0.000, E1   +74.438, E3 +157348.558}
SPL {X  -165.650, Y  +420.321, Z    +0.000, E1   +71.570, E3 +157437.212}
ENDSPLINE

SPLINE
SPL {X  -165.650, Y  +437.633, Z    +0.000, E1   +68.421, E3 +157452.960}
ENDSPLINE

SPLINE
SPL {X  -164.513, Y  +359.128, Z    +0.000, E1   +73.170, E3 +157463.194}
SPL {X  -163.967, Y  +354.944, Z    +0.000, E1   +72.327, E3 +157474.547}
SPL {X  -163.372, Y  +351.124, Z    +0.000, E1   +71.295, E3 +157487.139}
SPL {X  -162.653, Y  +347.134, Z    +0.000, E1   +70.371, E3 +157498.375}
SPL {X  -161.430, Y  +341.349, Z    +0.000, E1   +69.492, E3 +157510.449}
SPL {X  -160.389, Y  +337.084, Z    +0.000, E1   +68.301, E3 +157523.536}
SPL {X  -159.245, Y  +332.881, Z    +0.000, E1   +67.496, E3 +157533.196}
SPL {X  -157.072, Y  +325.885, Z    +0.000, E1   +67.020, E3 +157542.545}
SPL {X  -154.432, Y  +318.577, Z    +0.000, E1   +66.843, E3 +157549.750}
SPL {X  -151.047, Y  +310.495, Z    +0.000, E1   +66.593, E3 +157558.162}
SPL {X  -146.639, Y  +301.448, Z    +0.000, E1   +65.839, E3 +157570.371}
SPL {X  -142.469, Y  +293.987, Z    +0.000, E1   +65.133, E3 +157580.420}
SPL {X  -139.022, Y  +288.429, Z    +0.000, E1   +64.807, E3 +157586.618}
SPL {X  -136.717, Y  +284.968, Z    +0.000, E1   +64.044, E3 +157593.211}
SPL {X  -133.061, Y  +279.835, Z    +0.000, E1   +64.204, E3 +157596.624}
SPL {X  -118.927, Y  +263.191, Z    +0.000, E1   +67.951, E3 +157592.637}
SPL {X   -76.819, Y  +231.739, Z    +0.000, E1   +54.834, E3 +157770.643}
ENDSPLINE

SPLINE
SPL {X  -140.879, Y  +291.363, Z    +0.000, E1   +48.273, E3 +157878.084}
SPL {X  -158.845, Y  +331.507, Z    +0.000, E1   +33.834, E3 +157887.419}
SPL {X  -164.164, Y  +356.358, Z    +0.000, E1   +18.707, E3 +157883.741}
SPL {X  -165.341, Y  +368.384, Z    +0.000, E1   +10.076, E3 +157884.486}
SPL {X  -165.648, Y  +377.641, Z    +0.000, E1    +2.653, E3 +157883.836}
SPL {X  -165.650, Y  +380.500, Z    +0.000, E1    -0.000, E3 +157882.867}
SPL {X  -165.650, Y  +381.694, Z    +0.000, E1    -1.679, E3 +157882.269}
SPL {X  -165.650, Y  +384.595, Z    +0.000, E1    -6.546, E3 +157882.131}
SPL {X  -165.650, Y  +389.276, Z    +0.000, E1   -15.245, E3 +157881.639}
SPL {X  -165.650, Y  +395.801, Z    +0.000, E1   -28.236, E3 +157881.266}
SPL {X  -165.650, Y  +403.802, Z    +0.000, E1   -41.748, E3 +157881.087}
SPL {X  -165.650, Y  +419.045, Z    +0.000, E1   -60.641, E3 +157878.408}
SPL {X  -165.650, Y  +474.102, Z    +0.000, E1   -73.446, E3 +157890.191}
SPL {X  -165.650, Y  +640.142, Z    +0.000, E1   -72.635, E3 +157975.476}
ENDSPLINE

SPLINE
SPL {X  -165.650, Y  +612.217, Z    +0.000, E1   -68.647, E3 +157991.401}
ENDSPLINE

SPLINE
SPL {X  -165.650, Y  +623.643, Z    +0.000, E1   -68.543, E3 +158001.498}
SPL {X  -165.650, Y  +635.985, Z    +0.000, E1   -68.274, E3 +158013.876}
SPL {X  -165.650, Y  +656.072, Z    +0.000, E1   -68.403, E3 +158029.171}
SPL {X  -165.650, Y  +673.246, Z    +0.000, E1   -68.189, E3 +158044.926}
SPL {X  -164.760, Y  +692.647, Z    +0.000, E1   -68.400, E3 +158058.891}
SPL {X  -163.763, Y  +700.430, Z    +0.000, E1   -67.939, E3 +158068.914}
SPL {X  -161.478, Y  +712.444, Z    +0.000, E1   -67.895, E3 +158079.269}
SPL {X  -157.774, Y  +725.970, Z    +0.000, E1   -67.383, E3 +158094.271}
SPL {X  -153.458, Y  +737.875, Z    +0.000, E1   -66.902, E3 +158107.346}
SPL {X  -149.433, Y  +746.982, Z    +0.000, E1   -66.131, E3 +158119.977}
SPL {X  -144.642, Y  +756.238, Z    +0.000, E1   -65.678, E3 +158130.208}
SPL {X  -141.719, Y  +761.265, Z    +0.000, E1   -65.117, E3 +158137.341}
SPL {X  -139.420, Y  +764.954, Z    +0.000, E1   -64.577, E3 +158143.204}
SPL {X  -136.483, Y  +769.374, Z    +0.000, E1   -64.163, E3 +158148.859}
SPL {X  -133.523, Y  +773.539, Z    +0.000, E1   -63.962, E3 +158153.127}
SPL {X  -125.028, Y  +784.164, Z    +0.000, E1   -66.760, E3 +158149.203}
SPL {X   -71.589, Y  +824.882, Z    +0.000, E1   -56.415, E3 +158276.268}
ENDSPLINE

SPLINE
SPL {X  -127.072, Y  +781.767, Z    +0.000, E1   -54.186, E3 +158439.240}
SPL {X  -150.680, Y  +744.314, Z    +0.000, E1   -44.608, E3 +158450.196}
SPL {X  -162.376, Y  +708.273, Z    +0.000, E1   -25.870, E3 +158442.320}
SPL {X  -165.092, Y  +689.091, Z    +0.000, E1   -12.938, E3 +158443.739}
SPL {X  -165.629, Y  +678.122, Z    +0.000, E1    -4.178, E3 +158442.886}
SPL {X  -165.650, Y  +673.539, Z    +0.000, E1    -0.057, E3 +158441.984}
SPL {X  -165.650, Y  +671.359, Z    +0.000, E1    +3.116, E3 +158441.341}
SPL {X  -165.650, Y  +667.465, Z    +0.000, E1   +10.413, E3 +158441.135}
SPL {X  -165.650, Y  +662.220, Z    +0.000, E1   +20.600, E3 +158440.827}
SPL {X  -165.650, Y  +652.464, Z    +0.000, E1   +39.379, E3 +158439.774}
SPL {X  -165.650, Y  +636.657, Z    +0.000, E1   +60.410, E3 +158437.063}
SPL {X  -165.650, Y  +613.310, Z    +0.000, E1   +72.038, E3 +158437.422}
SPL {X  -165.650, Y  +568.914, Z    +0.000, E1   +74.438, E3 +158452.007}
SPL {X  -165.650, Y  +420.321, Z    +0.000, E1   +71.570, E3 +158540.660}
ENDSPLINE

SPLINE
SPL {X  -165.650, Y  +437.633, Z    +0.000, E1   +68.421, E3 +158556.408}
ENDSPLINE

SPLINE
SPL {X  -164.513, Y  +359.128, Z    +0.000, E1   +73.170, E3 +158566.642}
SPL {X  -163.967, Y  +354.944, Z    +0.000, E1   +72.327, E3 +158577.995}
SPL {X  -163.372, Y  +351.124, Z    +0.000, E1   +71.295, E3 +158590.587}
SPL {X  -162.653, Y  +347.134, Z    +0.000, E1   +70.371, E3 +158601.823}
SPL {X  -161.430, Y  +341.349, Z    +0.000, E1   +69.492, E3 +158613.897}
SPL {X  -160.389, Y  +337.084, Z    +0.000, E1   +68.301, E3 +158626.984}
SPL {X  -159.245, Y  +332.881, Z    +0.000, E1   +67.496, E3 +158636.644}
SPL {X  -157.072, Y  +325.885, Z    +0.000, E1   +67.020, E3 +158645.993}
SPL {X  -154.432, Y  +318.577, Z    +0.000, E1   +66.843, E3 +158653.198}
SPL {X  -151.047, Y  +310.495, Z    +0.000, E1   +66.593, E3 +158661.610}
SPL {X  -146.639, Y  +301.448, Z    +0.000, E1   +65.839, E3 +158673.820}
SPL {X  -142.469, Y  +293.987, Z    +0.000, E1   +65.133, E3 +158683.868}
SPL {X  -139.022, Y  +288.429, Z    +0.000, E1   +64.807, E3 +158690.067}
SPL {X  -136.717, Y  +284.968, Z    +0.000, E1   +64.044, E3 +158696.659}
SPL {X  -133.061, Y  +279.835, Z    +0.000, E1   +64.204, E3 +158700.073}
SPL {X  -118.927, Y  +263.191, Z    +0.000, E1   +67.951, E3 +158696.085}
SPL {X   -76.819, Y  +231.739, Z    +0.000, E1   +54.834, E3 +158874.091}
ENDSPLINE

SPLINE
SPL {X  -140.879, Y  +291.363, Z    +0.000, E1   +48.273, E3 +158981.532}
SPL {X  -158.845, Y  +331.507, Z    +0.000, E1   +33.834, E3 +158990.867}
SPL {X  -164.164, Y  +356.358, Z    +0.000, E1   +18.707, E3 +158987.190}
SPL {X  -165.341, Y  +368.384, Z    +0.000, E1   +10.076, E3 +158987.934}
SPL {X  -165.648, Y  +377.641, Z    +0.000, E1    +2.653, E3 +158987.285}
SPL {X  -165.650, Y  +380.500, Z    +0.000, E1    -0.000, E3 +158986.315}
SPL {X  -165.650, Y  +381.694, Z    +0.000, E1    -1.679, E3 +158985.717}
SPL {X  -165.650, Y  +384.595, Z    +0.000, E1    -6.546, E3 +158985.579}
SPL {X  -165.650, Y  +389.276, Z    +0.000, E1   -15.245, E3 +158985.087}
SPL {X  -165.650, Y  +395.801, Z    +0.000, E1   -28.236, E3 +158984.714}
SPL {X  -165.650, Y  +403.802, Z    +0.000, E1   -41.748, E3 +158984.535}
SPL {X  -165.650, Y  +419.045, Z    +0.000, E1   -60.641, E3 +158981.856}
SPL {X  -165.650, Y  +474.102, Z    +0.000, E1   -73.446, E3 +158993.640}
SPL {X  -165.650, Y  +640.142, Z    +0.000, E1   -72.635, E3 +159078.924}
ENDSPLINE

SPLINE
SPL {X  -165.650, Y  +612.217, Z    +0.000, E1   -68.647, E3 +159094.850}
ENDSPLINE

SPLINE
SPL {X  -165.650, Y  +623.643, Z    +0.000, E1   -68.543, E3 +159104.946}
SPL {X  -165.650, Y  +635.985, Z    +0.000, E1   -68.274, E3 +159117.325}
SPL {X  -165.650, Y  +656.072, Z    +0.000, E1   -68.403, E3 +159132.619}
SPL {X  -165.650, Y  +673.246, Z    +0.000, E1   -68.189, E3 +159148.374}
SPL {X  -164.760, Y  +692.647, Z    +0.000, E1   -68.400, E3 +159162.340}
SPL {X  -162.986, Y  +705.089, Z    +0.000, E1   -67.915, E3 +159176.551}
SPL {X  -159.812, Y  +719.091, Z    +0.000, E1   -67.711, E3 +159189.550}
SPL {X  -156.969, Y  +728.420, Z    +0.000, E1   -67.278, E3 +159200.333}
SPL {X  -153.458, Y  +737.875, Z    +0.000, E1   -66.902, E3 +159210.794}
SPL {X  -149.433, Y  +746.982, Z    +0.000, E1   -66.131, E3 +159223.425}
SPL {X  -144.642, Y  +756.238, Z    +0.000, E1   -65.678, E3 +159233.656}
SPL {X  -140.398, Y  +763.411, Z    +0.000, E1   -64.853, E3 +159244.132}
SPL {X  -135.180, Y  +771.240, Z    +0.000, E1   -64.104, E3 +159254.181}
SPL {X  -125.028, Y  +784.164, Z    +0.000, E1   -66.760, E3 +159252.651}
SPL {X   -71.589, Y  +824.882, Z    +0.000, E1   -56.415, E3 +159379.716}
ENDSPLINE

SPLINE
SPL {X  -127.072, Y  +781.767, Z    +0.000, E1   -54.186, E3 +159542.688}
SPL {X  -150.680, Y  +744.314, Z    +0.000, E1   -44.608, E3 +159553.645}
SPL {X  -162.376, Y  +708.273, Z    +0.000, E1   -25.870, E3 +159545.768}
SPL {X  -165.092, Y  +689.091, Z    +0.000, E1   -12.938, E3 +159547.187}
SPL {X  -165.629, Y  +678.122, Z    +0.000, E1    -4.178, E3 +159546.334}
SPL {X  -165.650, Y  +673.539, Z    +0.000, E1    -0.057, E3 +159545.432}
SPL {X  -165.650, Y  +671.359, Z    +0.000, E1    +3.116, E3 +159544.789}
SPL {X  -165.650, Y  +665.277, Z    +0.000, E1   +14.409, E3 +159544.434}
SPL {X  -165.650, Y  +659.573, Z    +0.000, E1   +26.182, E3 +159544.182}
SPL {X  -165.650, Y  +652.464, Z    +0.000, E1   +39.379, E3 +159543.223}
SPL {X  -165.650, Y  +634.871, Z    +0.000, E1   +61.762, E3 +159540.455}
SPL {X  -165.650, Y  +574.769, Z    +0.000, E1   +74.441, E3 +159553.103}
SPL {X  -165.650, Y  +420.321, Z    +0.000, E1   +71.570, E3 +159644.108}
ENDSPLINE

SPLINE
SPL {X  -165.650, Y  +437.633, Z    +0.000, E1   +68.421, E3 +159659.857}
ENDSPLINE

SPLINE
SPL {X  -164.513, Y  +359.128, Z    +0.000, E1   +73.170, E3 +159670.090}
SPL {X  -163.967, Y  +354.944, Z    +0.000, E1   +72.327, E3 +159681.443}
SPL {X  -163.372, Y  +351.124, Z    +0.000, E1   +71.295, E3 +159694.036}
SPL {X  -162.653, Y  +347.134, Z    +0.000, E1   +70.371, E3 +159705.271}
SPL {X  -161.430, Y  +341.349, Z    +0.000, E1   +69.492, E3 +159717.345}
SPL {X  -160.389, Y  +337.084, Z    +0.000, E1   +68.301, E3 +159730.433}
SPL {X  -158.795, Y  +331.340, Z    +0.000, E1   +67.291, E3 +159743.119}
SPL {X  -155.058, Y  +320.218, Z    +0.000, E1   +66.982, E3 +159754.425}
SPL {X  -151.047, Y  +310.495, Z    +0.000, E1   +66.593, E3 +159765.058}
SPL {X  -148.187, Y  +304.469, Z    +0.000, E1   +66.029, E3 +159773.437}
SPL {X  -145.703, Y  +299.692, Z    +0.000, E1   +65.663, E3 +159779.604}
SPL {X  -142.469, Y  +293.987, Z    +0.000, E1   +65.133, E3 +159787.316}
SPL {X  -139.022, Y  +288.429, Z    +0.000, E1   +64.807, E3 +159793.515}
SPL {X  -136.717, Y  +284.968, Z    +0.000, E1   +64.044, E3 +159800.107}
SPL {X  -133.061, Y  +279.835, Z    +0.000, E1   +64.204, E3 +159803.521}
SPL {X  -118.927, Y  +263.191, Z    +0.000, E1   +67.951, E3 +159799.533}
SPL {X   -76.819, Y  +231.739, Z    +0.000, E1   +54.834, E3 +159977.539}
ENDSPLINE

SPLINE
SPL {X  -140.879, Y  +291.363, Z    +0.000, E1   +48.273, E3 +160084.981}
SPL {X  -155.054, Y  +320.205, Z    +0.000, E1   +39.591, E3 +160097.432}
SPL {X  -160.978, Y  +339.437, Z    +0.000, E1   +29.257, E3 +160092.062}
SPL {X  -164.164, Y  +356.358, Z    +0.000, E1   +18.707, E3 +160090.638}
SPL {X  -165.519, Y  +371.910, Z    +0.000, E1    +7.409, E3 +160091.047}
SPL {X  -165.650, Y  +380.329, Z    +0.000, E1    +0.239, E3 +160089.893}
SPL {X  -165.650, Y  +381.694, Z    +0.000, E1    -1.679, E3 +160089.165}
SPL {X  -165.650, Y  +384.595, Z    +0.000, E1    -6.546, E3 +160089.027}
SPL {X  -165.650, Y  +389.276, Z    +0.000, E1   -15.245, E3 +160088.535}
SPL {X  -165.650, Y  +395.801, Z    +0.000, E1   -28.236, E3 +160088.163}
SPL {X  -165.650, Y  +403.802, Z    +0.000, E1   -41.748, E3 +160087.984}
SPL {X  -165.650, Y  +418.088, Z    +0.000, E1   -59.974, E3 +160085.256}
SPL {X  -165.650, Y  +461.994, Z    +0.000, E1   -72.657, E3 +160093.394}
SPL {X  -165.650, Y  +492.072, Z    +0.000, E1   -73.925, E3 +160103.496}
SPL {X  -165.650, Y  +637.039, Z    +0.000, E1   -73.842, E3 +160170.161}
ENDSPLINE

SPLINE
SPL {X  -165.650, Y  +617.598, Z    +0.000, E1   -69.273, E3 +160197.228}
ENDSPLINE

SPLINE
SPL {X  -165.650, Y  +623.643, Z    +0.000, E1   -68.543, E3 +160208.394}
SPL {X  -165.650, Y  +635.985, Z    +0.000, E1   -68.274, E3 +160220.773}
SPL {X  -165.650, Y  +647.687, Z    +0.000, E1   -68.151, E3 +160231.273}
SPL {X  -165.650, Y  +665.917, Z    +0.000, E1   -68.414, E3 +160244.032}
SPL {X  -165.417, Y  +684.287, Z    +0.000, E1   -68.467, E3 +160258.329}
SPL {X  -164.268, Y  +696.853, Z    +0.000, E1   -68.071, E3 +160271.959}
SPL {X  -162.443, Y  +707.938, Z    +0.000, E1   -67.853, E3 +160282.693}
SPL {X  -159.812, Y  +719.091, Z    +0.000, E1   -67.711, E3 +160292.999}
SPL {X  -156.969, Y  +728.420, Z    +0.000, E1   -67.278, E3 +160303.781}
SPL {X  -154.751, Y  +734.593, Z    +0.000, E1   -66.864, E3 +160311.762}
SPL {X  -151.443, Y  +742.618, Z    +0.000, E1   -66.527, E3 +160320.757}
SPL {X  -148.198, Y  +749.508, Z    +0.000, E1   -66.065, E3 +160329.238}
SPL {X  -144.642, Y  +756.238, Z    +0.000, E1   -65.678, E3 +160337.104}
SPL {X  -140.398, Y  +763.411, Z    +0.000, E1   -64.853, E3 +160347.580}
SPL {X  -135.180, Y  +771.240, Z    +0.000, E1   -64.104, E3 +160357.630}
SPL {X  -125.028, Y  +784.164, Z    +0.000, E1   -66.760, E3 +160356.100}
SPL {X   -74.840, Y  +823.280, Z    +0.000, E1   -57.857, E3 +160456.632}
SPL {X   -70.065, Y  +825.603, Z    +0.000, E1   -55.379, E3 +160516.934}
ENDSPLINE

SPLINE
SPL {X  -127.072, Y  +781.767, Z    +0.000, E1   -54.186, E3 +160646.137}
SPL {X  -150.680, Y  +744.314, Z    +0.000, E1   -44.608, E3 +160657.093}
SPL {X  -162.376, Y  +708.273, Z    +0.000, E1   -25.870, E3 +160649.217}
SPL {X  -165.092, Y  +689.091, Z    +0.000, E1   -12.938, E3 +160650.635}
SPL {X  -165.629, Y  +678.122, Z    +0.000, E1    -4.178, E3 +160649.783}
SPL {X  -165.650, Y  +673.539, Z    +0.000, E1    -0.057, E3 +160648.880}
SPL {X  -165.650, Y  +672.623, Z    +0.000, E1    +1.276, E3 +160648.360}
SPL {X  -165.650, Y  +669.039, Z    +0.000, E1    +7.218, E3 +160648.086}
SPL {X  -165.650, Y  +662.220, Z    +0.000, E1   +20.600, E3 +160647.723}
SPL {X  -165.650, Y  +652.464, Z    +0.000, E1   +39.379, E3 +160646.671}
SPL {X  -165.650, Y  +634.871, Z    +0.000, E1   +61.762, E3 +160643.904}
SPL {X  -165.650, Y  +574.769, Z    +0.000, E1   +74.441, E3 +160656.552}
SPL {X  -165.650, Y  +420.321, Z    +0.000, E1   +71.570, E3 +160747.557}
ENDSPLINE

SPLINE
SPL {X  -165.650, Y  +437.633, Z    +0.000, E1   +68.421, E3 +160763.305}
ENDSPLINE

SPLINE
SPL {X  -164.513, Y  +359.128, Z    +0.000, E1   +73.170, E3 +160773.538}
SPL {X  -163.967, Y  +354.944, Z    +0.000, E1   +72.327, E3 +160784.892}
SPL {X  -163.571, Y  +352.336, Z    +0.000, E1   +71.524, E3 +160794.310}
SPL {X  -162.836, Y  +348.099, Z    +0.000, E1   +70.646, E3 +160805.784}
SPL {X  -161.430, Y  +341.349, Z    +0.000, E1   +69.492, E3 +160820.794}
SPL {X  -160.389, Y  +337.084, Z    +0.000, E1   +68.301, E3 +160833.881}
SPL {X  -159.245, Y  +332.881, Z    +0.000, E1   +67.496, E3 +160843.541}
SPL {X  -157.072, Y  +325.885, Z    +0.000, E1   +67.020, E3 +160852.890}
SPL {X  -154.432, Y  +318.577, Z    +0.000, E1   +66.843, E3 +160860.095}
SPL {X  -151.047, Y  +310.495, Z    +0.000, E1   +66.593, E3 +160868.507}
SPL {X  -146.639, Y  +301.448, Z    +0.000, E1   +65.839, E3 +160880.716}
SPL {X  -142.469, Y  +293.987, Z    +0.000, E1   +65.133, E3 +160890.765}
SPL {X  -139.022, Y  +288.429, Z    +0.000, E1   +64.807, E3 +160896.963}
SPL {X  -136.717, Y  +284.968, Z    +0.000, E1   +64.044, E3 +160903.556}
SPL {X  -133.061, Y  +279.835, Z    +0.000, E1   +64.204, E3 +160906.969}
SPL {X  -118.927, Y  +263.191, Z    +0.000, E1   +67.951, E3 +160902.982}
SPL {X   -76.819, Y  +231.739, Z    +0.000, E1   +54.834, E3 +161080.988}
ENDSPLINE

SPLINE
SPL {X  -140.879, Y  +291.363, Z    +0.000, E1   +48.273, E3 +161188.429}
SPL {X  -158.845, Y  +331.507, Z    +0.000, E1   +33.834, E3 +161197.764}
SPL {X  -164.164, Y  +356.358, Z    +0.000, E1   +18.707, E3 +161194.086}
SPL {X  -165.341, Y  +368.384, Z    +0.000, E1   +10.076, E3 +161194.831}
SPL {X  -165.648, Y  +377.641, Z    +0.000, E1    +2.653, E3 +161194.181}
SPL {X  -165.650, Y  +380.939, Z    +0.000, E1    -0.407, E3 +161192.992}
SPL {X  -165.650, Y  +385.900, Z    +0.000, E1    -8.711, E3 +161192.436}
SPL {X  -165.650, Y  +390.854, Z    +0.000, E1   -18.692, E3 +161191.612}
SPL {X  -165.650, Y  +395.801, Z    +0.000, E1   -28.236, E3 +161191.611}
SPL {X  -165.650, Y  +403.802, Z    +0.000, E1   -41.748, E3 +161191.432}
SPL {X  -165.650, Y  +418.088, Z    +0.000, E1   -59.974, E3 +161188.704}
SPL {X  -165.650, Y  +461.994, Z    +0.000, E1   -72.657, E3 +161196.842}
SPL {X  -165.650, Y  +492.072, Z    +0.000, E1   -73.925, E3 +161206.944}
SPL {X  -165.650, Y  +640.142, Z    +0.000, E1   -72.635, E3 +161285.821}
ENDSPLINE

SPLINE
SPL {X  -165.650, Y  +612.217, Z    +0.000, E1   -68.647, E3 +161301.746}
ENDSPLINE

SPLINE
SPL {X  -165.650, Y  +623.643, Z    +0.000, E1   -68.543, E3 +161311.843}
SPL {X  -165.650, Y  +635.985, Z    +0.000, E1   -68.274, E3 +161324.221}
SPL {X  -165.650, Y  +647.687, Z    +0.000, E1   -68.151, E3 +161334.721}
SPL {X  -165.650, Y  +665.917, Z    +0.000, E1   -68.414, E3 +161347.481}
SPL {X  -165.417, Y  +684.287, Z    +0.000, E1   -68.467, E3 +161361.778}
SPL {X  -164.655, Y  +693.631, Z    +0.000, E1   -68.130, E3 +161372.129}
SPL {X  -162.986, Y  +705.089, Z    +0.000, E1   -67.915, E3 +161383.448}
SPL {X  -160.378, Y  +716.957, Z    +0.000, E1   -67.874, E3 +161393.268}
SPL {X  -157.774, Y  +725.970, Z    +0.000, E1   -67.383, E3 +161404.616}
SPL {X  -153.458, Y  +737.875, Z    +0.000, E1   -66.902, E3 +161417.691}
SPL {X  -150.971, Y  +743.674, Z    +0.000, E1   -66.152, E3 +161427.348}
SPL {X  -148.198, Y  +749.508, Z    +0.000, E1   -66.065, E3 +161432.686}
SPL {X  -144.642, Y  +756.238, Z    +0.000, E1   -65.678, E3 +161440.552}
SPL {X  -140.398, Y  +763.411, Z    +0.000, E1   -64.853, E3 +161451.028}
SPL {X  -135.180, Y  +771.240, Z    +0.000, E1   -64.104, E3 +161461.078}
SPL {X  -125.028, Y  +784.164, Z    +0.000, E1   -66.760, E3 +161459.548}
SPL {X   -71.589, Y  +824.882, Z    +0.000, E1   -56.415, E3 +161586.613}
ENDSPLINE

SPLINE
SPL {X  -127.072, Y  +781.767, Z    +0.000, E1   -54.186, E3 +161749.585}
SPL {X  -150.680, Y  +744.314, Z    +0.000, E1   -44.608, E3 +161760.541}
SPL {X  -162.376, Y  +708.273, Z    +0.000, E1   -25.870, E3 +161752.665}
SPL {X  -165.092, Y  +689.091, Z    +0.000, E1   -12.938, E3 +161754.084}
SPL {X  -165.629, Y  +678.122, Z    +0.000, E1    -4.178, E3 +161753.231}
SPL {X  -165.650, Y  +673.539, Z    +0.000, E1    -0.057, E3 +161752.329}
SPL {X  -165.650, Y  +671.359, Z    +0.000, E1    +3.116, E3 +161751.685}
SPL {X  -165.650, Y  +665.277, Z    +0.000, E1   +14.409, E3 +161751.330}
SPL {X  -165.650, Y  +656.188, Z    +0.000, E1   +32.567, E3 +161750.507}
SPL {X  -165.650, Y  +648.712, Z    +0.000, E1   +45.195, E3 +161750.129}
SPL {X  -165.650, Y  +636.657, Z    +0.000, E1   +60.410, E3 +161747.407}
SPL {X  -165.650, Y  +613.310, Z    +0.000, E1   +72.038, E3 +161747.767}
SPL {X  -165.650, Y  +568.914, Z    +0.000, E1   +74.438, E3 +161762.351}
SPL {X  -165.650, Y  +420.321, Z    +0.000, E1   +71.570, E3 +161851.005}
ENDSPLINE

SPLINE
SPL {X  -165.650, Y  +437.633, Z    +0.000, E1   +68.421, E3 +161866.753}
ENDSPLINE

SPLINE
SPL {X  -164.513, Y  +359.128, Z    +0.000, E1   +73.170, E3 +161876.987}
SPL {X  -163.967, Y  +354.944, Z    +0.000, E1   +72.327, E3 +161888.340}
SPL {X  -163.372, Y  +351.124, Z    +0.000, E1   +71.295, E3 +161900.932}
SPL {X  -162.653, Y  +347.134, Z    +0.000, E1   +70.371, E3 +161912.168}
SPL {X  -161.451, Y  +341.438, Z    +0.000, E1   +69.889, E3 +161920.487}
SPL {X  -161.195, Y  +340.340, Z    +0.000, E1   +68.690, E3 +161931.708}
SPL {X  -159.328, Y  +333.173, Z    +0.000, E1   +67.752, E3 +161944.928}
SPL {X  -158.153, Y  +329.228, Z    +0.000, E1   +66.894, E3 +161954.484}
SPL {X  -154.229, Y  +318.056, Z    +0.000, E1   +66.925, E3 +161963.620}
SPL {X  -149.308, Y  +306.758, Z    +0.000, E1   +66.321, E3 +161976.826}
SPL {X  -145.703, Y  +299.692, Z    +0.000, E1   +65.663, E3 +161986.500}
SPL {X  -142.469, Y  +293.987, Z    +0.000, E1   +65.133, E3 +161994.213}
SPL {X  -139.022, Y  +288.429, Z    +0.000, E1   +64.807, E3 +162000.412}
SPL {X  -136.717, Y  +284.968, Z    +0.000, E1   +64.044, E3 +162007.004}
SPL {X  -133.061, Y  +279.835, Z    +0.000, E1   +64.204, E3 +162010.418}
SPL {X  -118.927, Y  +263.191, Z    +0.000, E1   +67.951, E3 +162006.430}
SPL {X   -76.819, Y  +231.739, Z    +0.000, E1   +54.834, E3 +162184.436}
ENDSPLINE

SPLINE
SPL {X  -140.879, Y  +291.363, Z    +0.000, E1   +48.273, E3 +162291.877}
SPL {X  -158.845, Y  +331.507, Z    +0.000, E1   +33.834, E3 +162301.212}
SPL {X  -164.164, Y  +356.358, Z    +0.000, E1   +18.707, E3 +162297.535}
SPL {X  -165.341, Y  +368.384, Z    +0.000, E1   +10.076, E3 +162298.279}
SPL {X  -165.648, Y  +377.641, Z    +0.000, E1    +2.653, E3 +162297.630}
SPL {X  -165.650, Y  +380.939, Z    +0.000, E1    -0.407, E3 +162296.440}
SPL {X  -165.650, Y  +384.595, Z    +0.000, E1    -6.546, E3 +162295.924}
SPL {X  -165.650, Y  +389.276, Z    +0.000, E1   -15.245, E3 +162295.432}
SPL {X  -165.650, Y  +395.801, Z    +0.000, E1   -28.236, E3 +162295.059}
SPL {X  -165.650, Y  +403.802, Z    +0.000, E1   -41.748, E3 +162294.880}
SPL {X  -165.650, Y  +419.045, Z    +0.000, E1   -60.641, E3 +162292.201}
SPL {X  -165.650, Y  +474.102, Z    +0.000, E1   -73.446, E3 +162303.984}
SPL {X  -165.650, Y  +637.039, Z    +0.000, E1   -73.842, E3 +162377.058}
ENDSPLINE

SPLINE
SPL {X  -165.650, Y  +617.598, Z    +0.000, E1   -69.273, E3 +162404.124}
ENDSPLINE

SPLINE
SPL {X  -165.650, Y  +623.643, Z    +0.000, E1   -68.543, E3 +162415.291}
SPL {X  -165.650, Y  +635.985, Z    +0.000, E1   -68.274, E3 +162427.670}
SPL {X  -165.650, Y  +656.072, Z    +0.000, E1   -68.403, E3 +162442.964}
SPL {X  -165.650, Y  +673.246, Z    +0.000, E1   -68.189, E3 +162458.719}
SPL {X  -164.760, Y  +692.647, Z    +0.000, E1   -68.400, E3 +162472.685}
SPL {X  -162.986, Y  +705.089, Z    +0.000, E1   -67.915, E3 +162486.896}
SPL {X  -160.378, Y  +716.957, Z    +0.000, E1   -67.874, E3 +162496.716}
SPL {X  -157.774, Y  +725.970, Z    +0.000, E1   -67.383, E3 +162508.064}
SPL {X  -154.751, Y  +734.593, Z    +0.000, E1   -66.864, E3 +162518.658}
SPL {X  -151.443, Y  +742.618, Z    +0.000, E1   -66.527, E3 +162527.653}
SPL {X  -148.198, Y  +749.508, Z    +0.000, E1   -66.065, E3 +162536.134}
SPL {X  -144.642, Y  +756.238, Z    +0.000, E1   -65.678, E3 +162544.001}
SPL {X  -140.398, Y  +763.411, Z    +0.000, E1   -64.853, E3 +162554.477}
SPL {X  -135.180, Y  +771.240, Z    +0.000, E1   -64.104, E3 +162564.526}
SPL {X  -125.028, Y  +784.164, Z    +0.000, E1   -66.760, E3 +162562.996}
SPL {X   -71.589, Y  +824.882, Z    +0.000, E1   -56.415, E3 +162690.061}
ENDSPLINE

SPLINE
SPL {X  -127.072, Y  +781.767, Z    +0.000, E1   -54.186, E3 +162853.033}
SPL {X  -150.680, Y  +744.314, Z    +0.000, E1   -44.608, E3 +162863.990}
SPL {X  -162.376, Y  +708.273, Z    +0.000, E1   -25.870, E3 +162856.113}
SPL {X  -165.092, Y  +689.091, Z    +0.000, E1   -12.938, E3 +162857.532}
SPL {X  -165.629, Y  +678.122, Z    +0.000, E1    -4.178, E3 +162856.679}
SPL {X  -165.650, Y  +673.539, Z    +0.000, E1    -0.057, E3 +162855.777}
SPL {X  -165.650, Y  +671.359, Z    +0.000, E1    +3.116, E3 +162855.134}
SPL {X  -165.650, Y  +667.465, Z    +0.000, E1   +10.413, E3 +162854.928}
SPL {X  -165.650, Y  +662.220, Z    +0.000, E1   +20.600, E3 +162854.620}
SPL {X  -165.650, Y  +652.464, Z    +0.000, E1   +39.379, E3 +162853.568}
SPL {X  -165.650, Y  +636.657, Z    +0.000, E1   +60.410, E3 +162850.856}
SPL {X  -165.650, Y  +613.310, Z    +0.000, E1   +72.038, E3 +162851.215}
SPL {X  -165.650, Y  +568.914, Z    +0.000, E1   +74.438, E3 +162865.800}
SPL {X  -165.650, Y  +420.321, Z    +0.000, E1   +71.570, E3 +162954.453}
ENDSPLINE

SPLINE
SPL {X  -165.650, Y  +437.633, Z    +0.000, E1   +68.421, E3 +162970.201}
ENDSPLINE

SPLINE
SPL {X  -164.513, Y  +359.128, Z    +0.000, E1   +73.170, E3 +162980.435}
SPL {X  -163.967, Y  +354.944, Z    +0.000, E1   +72.327, E3 +162991.788}
SPL {X  -163.372, Y  +351.124, Z    +0.000, E1   +71.295, E3 +163004.381}
SPL {X  -162.653, Y  +347.134, Z    +0.000, E1   +70.371, E3 +163015.616}
SPL {X  -161.451, Y  +341.438, Z    +0.000, E1   +69.889, E3 +163023.935}
SPL {X  -161.444, Y  +341.410, Z    +0.000, E1   +69.001, E3 +163031.522}
SPL {X  -160.389, Y  +337.084, Z    +0.000, E1   +68.301, E3 +163040.777}
SPL {X  -158.795, Y  +331.340, Z    +0.000, E1   +67.291, E3 +163053.464}
SPL {X  -154.229, Y  +318.056, Z    +0.000, E1   +66.925, E3 +163067.068}
SPL {X  -149.308, Y  +306.758, Z    +0.000, E1   +66.321, E3 +163080.274}
SPL {X  -145.703, Y  +299.692, Z    +0.000, E1   +65.663, E3 +163089.949}
SPL {X  -142.469, Y  +293.987, Z    +0.000, E1   +65.133, E3 +163097.661}
SPL {X  -139.022, Y  +288.429, Z    +0.000, E1   +64.807, E3 +163103.860}
SPL {X  -136.717, Y  +284.968, Z    +0.000, E1   +64.044, E3 +163110.452}
SPL {X  -133.061, Y  +279.835, Z    +0.000, E1   +64.204, E3 +163113.866}
SPL {X  -118.927, Y  +263.191, Z    +0.000, E1   +67.951, E3 +163109.878}
SPL {X   -76.819, Y  +231.739, Z    +0.000, E1   +54.834, E3 +163287.884}
ENDSPLINE

SPLINE
SPL {X  -140.879, Y  +291.363, Z    +0.000, E1   +48.273, E3 +163395.326}
SPL {X  -158.845, Y  +331.507, Z    +0.000, E1   +33.834, E3 +163404.660}
SPL {X  -164.164, Y  +356.358, Z    +0.000, E1   +18.707, E3 +163400.983}
SPL {X  -165.341, Y  +368.384, Z    +0.000, E1   +10.076, E3 +163401.727}
SPL {X  -165.648, Y  +377.641, Z    +0.000, E1    +2.653, E3 +163401.078}
SPL {X  -165.650, Y  +380.500, Z    +0.000, E1    -0.000, E3 +163400.108}
SPL {X  -165.650, Y  +381.694, Z    +0.000, E1    -1.679, E3 +163399.510}
SPL {X  -165.650, Y  +384.595, Z    +0.000, E1    -6.546, E3 +163399.372}
SPL {X  -165.650, Y  +389.276, Z    +0.000, E1   -15.245, E3 +163398.880}
SPL {X  -165.650, Y  +395.801, Z    +0.000, E1   -28.236, E3 +163398.508}
SPL {X  -165.650, Y  +403.802, Z    +0.000, E1   -41.748, E3 +163398.328}
SPL {X  -165.650, Y  +419.045, Z    +0.000, E1   -60.641, E3 +163395.649}
SPL {X  -165.650, Y  +466.630, Z    +0.000, E1   -73.161, E3 +163404.777}
SPL {X  -165.650, Y  +492.072, Z    +0.000, E1   -73.925, E3 +163413.841}
SPL {X  -165.650, Y  +637.039, Z    +0.000, E1   -73.842, E3 +163480.506}
ENDSPLINE

SPLINE
SPL {X  -165.650, Y  +617.598, Z    +0.000, E1   -69.273, E3 +163507.573}
ENDSPLINE

SPLINE
SPL {X  -165.650, Y  +623.643, Z    +0.000, E1   -68.543, E3 +163518.739}
SPL {X  -165.650, Y  +635.985, Z    +0.000, E1   -68.274, E3 +163531.118}
SPL {X  -165.650, Y  +656.072, Z    +0.000, E1   -68.403, E3 +163546.412}
SPL {X  -165.650, Y  +669.180, Z    +0.000, E1   -68.170, E3 +163558.879}
SPL {X  -165.417, Y  +684.287, Z    +0.000, E1   -68.467, E3 +163568.674}
SPL {X  -164.268, Y  +696.853, Z    +0.000, E1   -68.071, E3 +163582.304}
SPL {X  -162.443, Y  +707.938, Z    +0.000, E1   -67.853, E3 +163593.038}
SPL {X  -159.812, Y  +719.091, Z    +0.000, E1   -67.711, E3 +163603.343}
SPL {X  -156.969, Y  +728.420, Z    +0.000, E1   -67.278, E3 +163614.126}
SPL {X  -154.751, Y  +734.593, Z    +0.000, E1   -66.864, E3 +163622.107}
SPL {X  -151.443, Y  +742.618, Z    +0.000, E1   -66.527, E3 +163631.101}
SPL {X  -148.198, Y  +749.508, Z    +0.000, E1   -66.065, E3 +163639.582}
SPL {X  -144.642, Y  +756.238, Z    +0.000, E1   -65.678, E3 +163647.449}
SPL {X  -140.398, Y  +763.411, Z    +0.000, E1   -64.853, E3 +163657.925}
SPL {X  -136.483, Y  +769.374, Z    +0.000, E1   -64.163, E3 +163666.100}
SPL {X  -133.523, Y  +773.539, Z    +0.000, E1   -63.962, E3 +163670.369}
SPL {X  -127.756, Y  +780.943, Z    +0.000, E1   -66.344, E3 +163665.963}
SPL {X  -118.855, Y  +790.884, Z    +0.000, E1   -67.633, E3 +163667.332}
SPL {X   -71.589, Y  +824.882, Z    +0.000, E1   -56.415, E3 +163793.509}
ENDSPLINE

SPLINE
SPL {X  -127.072, Y  +781.767, Z    +0.000, E1   -54.186, E3 +163956.481}
SPL {X  -150.680, Y  +744.314, Z    +0.000, E1   -44.608, E3 +163967.438}
SPL {X  -162.376, Y  +708.273, Z    +0.000, E1   -25.870, E3 +163959.561}
SPL {X  -165.092, Y  +689.091, Z    +0.000, E1   -12.938, E3 +163960.980}
SPL {X  -165.629, Y  +678.122, Z    +0.000, E1    -4.178, E3 +163960.127}
SPL {X  -165.650, Y  +673.539, Z    +0.000, E1    -0.057, E3 +163959.225}
SPL {X  -165.650, Y  +671.359, Z    +0.000, E1    +3.116, E3 +163958.582}
SPL {X  -165.650, Y  +665.277, Z    +0.000, E1   +14.409, E3 +163958.227}
SPL {X  -165.650, Y  +659.573, Z    +0.000, E1   +26.182, E3 +163957.975}
SPL {X  -165.650, Y  +652.464, Z    +0.000, E1   +39.379, E3 +163957.016}
SPL {X  -165.650, Y  +634.871, Z    +0.000, E1   +61.762, E3 +163954.248}
SPL {X  -165.650, Y  +574.769, Z    +0.000, E1   +74.441, E3 +163966.897}
SPL {X  -165.650, Y  +420.321, Z    +0.000, E1   +71.570, E3 +164057.901}
ENDSPLINE

SPLINE
SPL {X  -165.650, Y  +437.633, Z    +0.000, E1   +68.421, E3 +164073.650}
ENDSPLINE

SPLINE
SPL {X  -164.513, Y  +359.128, Z    +0.000, E1   +73.170, E3 +164083.883}
SPL {X  -163.967, Y  +354.944, Z    +0.000, E1   +72.327, E3 +164095.237}
SPL {X  -163.571, Y  +352.336, Z    +0.000, E1   +71.524, E3 +164104.655}
SPL {X  -162.836, Y  +348.099, Z    +0.000, E1   +70.646, E3 +164116.128}
SPL {X  -161.430, Y  +341.349, Z    +0.000, E1   +69.492, E3 +164131.138}
SPL {X  -160.389, Y  +337.084, Z    +0.000, E1   +68.301, E3 +164144.226}
SPL {X  -158.795, Y  +331.340, Z    +0.000, E1   +67.291, E3 +164156.912}
SPL {X  -155.058, Y  +320.218, Z    +0.000, E1   +66.982, E3 +164168.218}
SPL {X  -151.047, Y  +310.495, Z    +0.000, E1   +66.593, E3 +164178.852}
SPL {X  -146.639, Y  +301.448, Z    +0.000, E1   +65.839, E3 +164191.061}
SPL {X  -142.469, Y  +293.987, Z    +0.000, E1   +65.133, E3 +164201.110}
SPL {X  -139.022, Y  +288.429, Z    +0.000, E1   +64.807, E3 +164207.308}
SPL {X  -136.717, Y  +284.968, Z    +0.000, E1   +64.044, E3 +164213.900}
SPL {X  -133.061, Y  +279.835, Z    +0.000, E1   +64.204, E3 +164217.314}
SPL {X  -118.927, Y  +263.191, Z    +0.000, E1   +67.951, E3 +164213.326}
SPL {X   -76.819, Y  +231.739, Z    +0.000, E1   +54.834, E3 +164391.333}
ENDSPLINE

SPLINE
SPL {X  -140.879, Y  +291.363, Z    +0.000, E1   +48.273, E3 +164498.774}
SPL {X  -158.845, Y  +331.507, Z    +0.000, E1   +33.834, E3 +164508.109}
SPL {X  -164.164, Y  +356.358, Z    +0.000, E1   +18.707, E3 +164504.431}
SPL {X  -165.341, Y  +368.384, Z    +0.000, E1   +10.076, E3 +164505.175}
SPL {X  -165.648, Y  +377.641, Z    +0.000, E1    +2.653, E3 +164504.526}
SPL {X  -165.650, Y  +380.500, Z    +0.000, E1    -0.000, E3 +164503.557}
SPL {X  -165.650, Y  +381.694, Z    +0.000, E1    -1.679, E3 +164502.958}
SPL {X  -165.650, Y  +384.595, Z    +0.000, E1    -6.546, E3 +164502.820}
SPL {X  -165.650, Y  +389.276, Z    +0.000, E1   -15.245, E3 +164502.328}
SPL {X  -165.650, Y  +395.801, Z    +0.000, E1   -28.236, E3 +164501.956}
SPL {X  -165.650, Y  +403.802, Z    +0.000, E1   -41.748, E3 +164501.777}
SPL {X  -165.650, Y  +419.045, Z    +0.000, E1   -60.641, E3 +164499.098}
SPL {X  -165.650, Y  +474.102, Z    +0.000, E1   -73.446, E3 +164510.881}
SPL {X  -165.650, Y  +640.142, Z    +0.000, E1   -72.635, E3 +164596.166}
ENDSPLINE

SPLINE
SPL {X  -165.650, Y  +619.423, Z    +0.000, E1   -68.618, E3 +164618.363}
ENDSPLINE

SPLINE
SPL {X  -165.650, Y  +635.985, Z    +0.000, E1   -68.274, E3 +164634.566}
SPL {X  -165.650, Y  +647.687, Z    +0.000, E1   -68.151, E3 +164645.066}
SPL {X  -165.650, Y  +665.917, Z    +0.000, E1   -68.414, E3 +164657.825}
SPL {X  -165.417, Y  +684.287, Z    +0.000, E1   -68.467, E3 +164672.123}
SPL {X  -164.268, Y  +696.853, Z    +0.000, E1   -68.071, E3 +164685.752}
SPL {X  -161.478, Y  +712.444, Z    +0.000, E1   -67.895, E3 +164699.959}
SPL {X  -157.774, Y  +725.970, Z    +0.000, E1   -67.383, E3 +164714.960}
SPL {X  -154.751, Y  +734.593, Z    +0.000, E1   -66.864, E3 +164725.555}
SPL {X  -151.443, Y  +742.618, Z    +0.000, E1   -66.527, E3 +164734.550}
SPL {X  -146.969, Y  +751.920, Z    +0.000, E1   -66.066, E3 +164745.046}
SPL {X  -142.811, Y  +759.434, Z    +0.000, E1   -65.254, E3 +164755.895}
SPL {X  -139.420, Y  +764.954, Z    +0.000, E1   -64.577, E3 +164763.894}
SPL {X  -136.483, Y  +769.374, Z    +0.000, E1   -64.163, E3 +164769.549}
SPL {X  -133.523, Y  +773.539, Z    +0.000, E1   -63.962, E3 +164773.817}
SPL {X  -125.028, Y  +784.164, Z    +0.000, E1   -66.760, E3 +164769.893}
SPL {X   -71.589, Y  +824.882, Z    +0.000, E1   -56.415, E3 +164896.958}
ENDSPLINE

SPLINE
SPL {X  -127.072, Y  +781.767, Z    +0.000, E1   -54.186, E3 +165059.930}
SPL {X  -150.680, Y  +744.314, Z    +0.000, E1   -44.608, E3 +165070.886}
SPL {X  -162.376, Y  +708.273, Z    +0.000, E1   -25.870, E3 +165063.010}
SPL {X  -165.092, Y  +689.091, Z    +0.000, E1   -12.938, E3 +165064.429}
SPL {X  -165.629, Y  +678.122, Z    +0.000, E1    -4.178, E3 +165063.576}
SPL {X  -165.650, Y  +673.539, Z    +0.000, E1    -0.057, E3 +165062.673}
SPL {X  -165.650, Y  +671.359, Z    +0.000, E1    +3.116, E3 +165062.030}
SPL {X  -165.650, Y  +665.277, Z    +0.000, E1   +14.409, E3 +165061.675}
SPL {X  -165.650, Y  +659.573, Z    +0.000, E1   +26.182, E3 +165061.423}
SPL {X  -165.650, Y  +652.464, Z    +0.000, E1   +39.379, E3 +165060.464}
SPL {X  -165.650, Y  +634.871, Z    +0.000, E1   +61.762, E3 +165057.697}
SPL {X  -165.650, Y  +574.769, Z    +0.000, E1   +74.441, E3 +165070.345}
SPL {X  -165.650, Y  +420.321, Z    +0.000, E1   +71.570, E3 +165161.350}
ENDSPLINE

SPLINE
SPL {X  -165.650, Y  +437.633, Z    +0.000, E1   +68.421, E3 +165177.098}
ENDSPLINE

SPLINE
SPL {X  -164.513, Y  +359.128, Z    +0.000, E1   +73.170, E3 +165187.332}
SPL {X  -163.967, Y  +354.944, Z    +0.000, E1   +72.327, E3 +165198.685}
SPL {X  -163.372, Y  +351.124, Z    +0.000, E1   +71.295, E3 +165211.277}
SPL {X  -162.653, Y  +347.134, Z    +0.000, E1   +70.371, E3 +165222.512}
SPL {X  -161.430, Y  +341.349, Z    +0.000, E1   +69.492, E3 +165234.587}
SPL {X  -160.389, Y  +337.084, Z    +0.000, E1   +68.301, E3 +165247.674}
SPL {X  -158.795, Y  +331.340, Z    +0.000, E1   +67.291, E3 +165260.360}
SPL {X  -155.058, Y  +320.218, Z    +0.000, E1   +66.982, E3 +165271.666}
SPL {X  -151.047, Y  +310.495, Z    +0.000, E1   +66.593, E3 +165282.300}
SPL {X  -148.187, Y  +304.469, Z    +0.000, E1   +66.029, E3 +165290.679}
SPL {X  -145.703, Y  +299.692, Z    +0.000, E1   +65.663, E3 +165296.845}
SPL {X  -142.469, Y  +293.987, Z    +0.000, E1   +65.133, E3 +165304.558}
SPL {X  -139.022, Y  +288.429, Z    +0.000, E1   +64.807, E3 +165310.756}
SPL {X  -136.717, Y  +284.968, Z    +0.000, E1   +64.044, E3 +165317.349}
SPL {X  -133.061, Y  +279.835, Z    +0.000, E1   +64.204, E3 +165320.762}
SPL {X  -118.927, Y  +263.191, Z    +0.000, E1   +67.951, E3 +165316.775}
SPL {X   -76.819, Y  +231.739, Z    +0.000, E1   +54.834, E3 +165494.781}
ENDSPLINE

SPLINE
SPL {X  -140.879, Y  +291.363, Z    +0.000, E1   +48.273, E3 +165602.222}
SPL {X  -158.845, Y  +331.507, Z    +0.000, E1   +33.834, E3 +165611.557}
SPL {X  -164.164, Y  +356.358, Z    +0.000, E1   +18.707, E3 +165607.879}
SPL {X  -165.519, Y  +371.910, Z    +0.000, E1    +7.409, E3 +165608.288}
SPL {X  -165.650, Y  +380.329, Z    +0.000, E1    +0.239, E3 +165607.134}
SPL {X  -165.650, Y  +381.694, Z    +0.000, E1    -1.679, E3 +165606.407}
SPL {X  -165.650, Y  +384.595, Z    +0.000, E1    -6.546, E3 +165606.269}
SPL {X  -165.650, Y  +389.276, Z    +0.000, E1   -15.245, E3 +165605.777}
SPL {X  -165.650, Y  +395.801, Z    +0.000, E1   -28.236, E3 +165605.404}
SPL {X  -165.650, Y  +403.802, Z    +0.000, E1   -41.748, E3 +165605.225}
SPL {X  -165.650, Y  +418.088, Z    +0.000, E1   -59.974, E3 +165602.498}
SPL {X  -165.650, Y  +461.994, Z    +0.000, E1   -72.657, E3 +165610.635}
SPL {X  -165.650, Y  +492.072, Z    +0.000, E1   -73.925, E3 +165620.738}
SPL {X  -165.650, Y  +640.142, Z    +0.000, E1   -72.635, E3 +165699.614}
ENDSPLINE

SPLINE
SPL {X  -165.650, Y  +619.423, Z    +0.000, E1   -68.618, E3 +165721.811}
ENDSPLINE

SPLINE
SPL {X  -165.650, Y  +635.985, Z    +0.000, E1   -68.274, E3 +165738.014}
SPL {X  -165.650, Y  +647.687, Z    +0.000, E1   -68.151, E3 +165748.514}
SPL {X  -165.650, Y  +662.755, Z    +0.000, E1   -68.565, E3 +165757.181}
SPL {X  -165.650, Y  +673.246, Z    +0.000, E1   -68.189, E3 +165769.064}
SPL {X  -164.760, Y  +692.647, Z    +0.000, E1   -68.400, E3 +165783.029}
SPL {X  -163.763, Y  +700.430, Z    +0.000, E1   -67.939, E3 +165793.052}
SPL {X  -162.443, Y  +707.938, Z    +0.000, E1   -67.853, E3 +165799.934}
SPL {X  -159.812, Y  +719.091, Z    +0.000, E1   -67.711, E3 +165810.240}
SPL {X  -156.969, Y  +728.420, Z    +0.000, E1   -67.278, E3 +165821.022}
SPL {X  -154.751, Y  +734.593, Z    +0.000, E1   -66.864, E3 +165829.003}
SPL {X  -151.443, Y  +742.618, Z    +0.000, E1   -66.527, E3 +165837.998}
SPL {X  -148.198, Y  +749.508, Z    +0.000, E1   -66.065, E3 +165846.479}
SPL {X  -144.642, Y  +756.238, Z    +0.000, E1   -65.678, E3 +165854.345}
SPL {X  -140.398, Y  +763.411, Z    +0.000, E1   -64.853, E3 +165864.822}
SPL {X  -135.180, Y  +771.240, Z    +0.000, E1   -64.104, E3 +165874.871}
SPL {X  -125.028, Y  +784.164, Z    +0.000, E1   -66.760, E3 +165873.341}
SPL {X   -71.589, Y  +824.882, Z    +0.000, E1   -56.415, E3 +166000.406}
ENDSPLINE

SPLINE
SPL {X  -127.072, Y  +781.767, Z    +0.000, E1   -54.186, E3 +166163.378}
SPL {X  -150.680, Y  +744.314, Z    +0.000, E1   -44.608, E3 +166174.334}
SPL {X  -162.376, Y  +708.273, Z    +0.000, E1   -25.870, E3 +166166.458}
SPL {X  -165.092, Y  +689.091, Z    +0.000, E1   -12.938, E3 +166167.877}
SPL {X  -165.629, Y  +678.122, Z    +0.000, E1    -4.178, E3 +166167.024}
SPL {X  -165.650, Y  +673.290, Z    +0.000, E1    +0.167, E3 +166165.980}
SPL {X  -165.650, Y  +669.039, Z    +0.000, E1    +7.218, E3 +166165.327}
SPL {X  -165.650, Y  +662.220, Z    +0.000, E1   +20.600, E3 +166164.965}
SPL {X  -165.650, Y  +652.464, Z    +0.000, E1   +39.379, E3 +166163.912}
SPL {X  -165.650, Y  +634.871, Z    +0.000, E1   +61.762, E3 +166161.145}
SPL {X  -165.650, Y  +574.769, Z    +0.000, E1   +74.441, E3 +166173.793}
SPL {X  -165.650, Y  +420.321, Z    +0.000, E1   +71.570, E3 +166264.798}
ENDSPLINE

SPLINE
SPL {X  -165.650, Y  +437.633, Z    +0.000, E1   +68.421, E3 +166280.546}
ENDSPLINE

SPLINE
SPL {X  -164.513, Y  +359.128, Z    +0.000, E1   +73.170, E3 +166290.780}
SPL {X  -163.967, Y  +354.944, Z    +0.000, E1   +72.327, E3 +166302.133}
SPL {X  -163.372, Y  +351.124, Z    +0.000, E1   +71.295, E3 +166314.725}
SPL {X  -162.653, Y  +347.134, Z    +0.000, E1   +70.371, E3 +166325.961}
SPL {X  -161.430, Y  +341.349, Z    +0.000, E1   +69.492, E3 +166338.035}
SPL {X  -160.389, Y  +337.084, Z    +0.000, E1   +68.301, E3 +166351.122}
SPL {X  -159.245, Y  +332.881, Z    +0.000, E1   +67.496, E3 +166360.782}
SPL {X  -157.072, Y  +325.885, Z    +0.000, E1   +67.020, E3 +166370.131}
SPL {X  -154.432, Y  +318.577, Z    +0.000, E1   +66.843, E3 +166377.336}
SPL {X  -151.047, Y  +310.495, Z    +0.000, E1   +66.593, E3 +166385.748}
SPL {X  -148.187, Y  +304.469, Z    +0.000, E1   +66.029, E3 +166394.127}
SPL {X  -145.703, Y  +299.692, Z    +0.000, E1   +65.663, E3 +166400.293}
SPL {X  -142.469, Y  +293.987, Z    +0.000, E1   +65.133, E3 +166408.006}
SPL {X  -139.022, Y  +288.429, Z    +0.000, E1   +64.807, E3 +166414.205}
SPL {X  -136.717, Y  +284.968, Z    +0.000, E1   +64.044, E3 +166420.797}
SPL {X  -133.061, Y  +279.835, Z    +0.000, E1   +64.204, E3 +166424.211}
SPL {X  -118.927, Y  +263.191, Z    +0.000, E1   +67.951, E3 +166420.223}
SPL {X   -76.819, Y  +231.739, Z    +0.000, E1   +54.834, E3 +166598.229}
ENDSPLINE

SPLINE
SPL {X  -140.879, Y  +291.363, Z    +0.000, E1   +48.273, E3 +166705.670}
SPL {X  -155.054, Y  +320.205, Z    +0.000, E1   +39.591, E3 +166718.122}
SPL {X  -160.978, Y  +339.437, Z    +0.000, E1   +29.257, E3 +166712.751}
SPL {X  -164.164, Y  +356.358, Z    +0.000, E1   +18.707, E3 +166711.328}
SPL {X  -165.519, Y  +371.910, Z    +0.000, E1    +7.409, E3 +166711.737}
SPL {X  -165.650, Y  +380.329, Z    +0.000, E1    +0.239, E3 +166710.583}
SPL {X  -165.650, Y  +381.694, Z    +0.000, E1    -1.679, E3 +166709.855}
SPL {X  -165.650, Y  +384.595, Z    +0.000, E1    -6.546, E3 +166709.717}
SPL {X  -165.650, Y  +389.276, Z    +0.000, E1   -15.245, E3 +166709.225}
SPL {X  -165.650, Y  +395.801, Z    +0.000, E1   -28.236, E3 +166708.852}
SPL {X  -165.650, Y  +403.802, Z    +0.000, E1   -41.748, E3 +166708.673}
SPL {X  -165.650, Y  +419.045, Z    +0.000, E1   -60.641, E3 +166705.994}
SPL {X  -165.650, Y  +474.102, Z    +0.000, E1   -73.446, E3 +166717.778}
SPL {X  -165.650, Y  +640.142, Z    +0.000, E1   -72.635, E3 +166803.062}
ENDSPLINE

SPLINE
SPL {X  -165.650, Y  +612.217, Z    +0.000, E1   -68.647, E3 +166818.987}
ENDSPLINE

SPLINE
SPL {X  -165.650, Y  +623.643, Z    +0.000, E1   -68.543, E3 +166829.084}
SPL {X  -165.650, Y  +635.985, Z    +0.000, E1   -68.274, E3 +166841.463}
SPL {X  -165.650, Y  +647.687, Z    +0.000, E1   -68.151, E3 +166851.962}
SPL {X  -165.650, Y  +665.917, Z    +0.000, E1   -68.414, E3 +166864.722}
SPL {X  -165.417, Y  +684.287, Z    +0.000, E1   -68.467, E3 +166879.019}
SPL {X  -164.268, Y  +696.853, Z    +0.000, E1   -68.071, E3 +166892.648}
SPL {X  -162.443, Y  +707.938, Z    +0.000, E1   -67.853, E3 +166903.383}
SPL {X  -159.812, Y  +719.091, Z    +0.000, E1   -67.711, E3 +166913.688}
SPL {X  -156.969, Y  +728.420, Z    +0.000, E1   -67.278, E3 +166924.470}
SPL {X  -153.458, Y  +737.875, Z    +0.000, E1   -66.902, E3 +166934.932}
SPL {X  -149.433, Y  +746.982, Z    +0.000, E1   -66.131, E3 +166947.563}
SPL {X  -144.642, Y  +756.238, Z    +0.000, E1   -65.678, E3 +166957.794}
SPL {X  -140.398, Y  +763.411, Z    +0.000, E1   -64.853, E3 +166968.270}
SPL {X  -135.180, Y  +771.240, Z    +0.000, E1   -64.104, E3 +166978.319}
SPL {X  -125.028, Y  +784.164, Z    +0.000, E1   -66.760, E3 +166976.789}
SPL {X   -71.589, Y  +824.882, Z    +0.000, E1   -56.415, E3 +167103.854}
ENDSPLINE

SPLINE
SPL {X  -127.072, Y  +781.767, Z    +0.000, E1   -54.186, E3 +167266.826}
SPL {X  -150.680, Y  +744.314, Z    +0.000, E1   -44.608, E3 +167277.783}
SPL {X  -162.376, Y  +708.273, Z    +0.000, E1   -25.870, E3 +167269.906}
SPL {X  -165.092, Y  +689.091, Z    +0.000, E1   -12.938, E3 +167271.325}
SPL {X  -165.629, Y  +678.122, Z    +0.000, E1    -4.178, E3 +167270.472}
SPL {X  -165.650, Y  +673.539, Z    +0.000, E1    -0.057, E3 +167269.570}
SPL {X  -165.650, Y  +671.359, Z    +0.000, E1    +3.116, E3 +167268.927}
SPL {X  -165.650, Y  +665.277, Z    +0.000, E1   +14.409, E3 +167268.572}
SPL {X  -165.650, Y  +659.573, Z    +0.000, E1   +26.182, E3 +167268.320}
SPL {X  -165.650, Y  +652.464, Z    +0.000, E1   +39.379, E3 +167267.361}
SPL {X  -165.650, Y  +634.871, Z    +0.000, E1   +61.762, E3 +167264.593}
SPL {X  -165.650, Y  +574.769, Z    +0.000, E1   +74.441, E3 +167277.241}
SPL {X  -165.650, Y  +420.321, Z    +0.000, E1   +71.570, E3 +167368.246}
ENDSPLINE

SPLINE
SPL {X  -165.650, Y  +437.633, Z    +0.000, E1   +68.421, E3 +167383.995}
ENDSPLINE

SPLINE
SPL {X  -164.513, Y  +359.128, Z    +0.000, E1   +73.170, E3 +167394.228}
SPL {X  -163.967, Y  +354.944, Z    +0.000, E1   +72.327, E3 +167405.581}
SPL {X  -163.571, Y  +352.336, Z    +0.000, E1   +71.524, E3 +167414.999}
SPL {X  -162.836, Y  +348.099, Z    +0.000, E1   +70.646, E3 +167426.473}
SPL {X  -161.430, Y  +341.349, Z    +0.000, E1   +69.492, E3 +167441.483}
SPL {X  -160.389, Y  +337.084, Z    +0.000, E1   +68.301, E3 +167454.571}
SPL {X  -158.795, Y  +331.340, Z    +0.000, E1   +67.291, E3 +167467.257}
SPL {X  -155.058, Y  +320.218, Z    +0.000, E1   +66.982, E3 +167478.563}
SPL {X  -151.047, Y  +310.495, Z    +0.000, E1   +66.593, E3 +167489.196}
SPL {X  -146.639, Y  +301.448, Z    +0.000, E1   +65.839, E3 +167501.406}
SPL {X  -142.469, Y  +293.987, Z    +0.000, E1   +65.133, E3 +167511.454}
SPL {X  -139.022, Y  +288.429, Z    +0.000, E1   +64.807, E3 +167517.653}
SPL {X  -136.717, Y  +284.968, Z    +0.000, E1   +64.044, E3 +167524.245}
SPL {X  -133.061, Y  +279.835, Z    +0.000, E1   +64.204, E3 +167527.659}
SPL {X  -118.927, Y  +263.191, Z    +0.000, E1   +67.951, E3 +167523.671}
SPL {X   -76.819, Y  +231.739, Z    +0.000, E1   +54.834, E3 +167701.677}
ENDSPLINE

SPLINE
SPL {X  -140.879, Y  +291.363, Z    +0.000, E1   +48.273, E3 +167809.119}
SPL {X  -158.845, Y  +331.507, Z    +0.000, E1   +33.834, E3 +167818.453}
SPL {X  -164.164, Y  +356.358, Z    +0.000, E1   +18.707, E3 +167814.776}
SPL {X  -165.341, Y  +368.384, Z    +0.000, E1   +10.076, E3 +167815.520}
SPL {X  -165.648, Y  +377.641, Z    +0.000, E1    +2.653, E3 +167814.871}
SPL {X  -165.650, Y  +380.500, Z    +0.000, E1    -0.000, E3 +167813.901}
SPL {X  -165.650, Y  +381.694, Z    +0.000, E1    -1.679, E3 +167813.303}
SPL {X  -165.650, Y  +384.595, Z    +0.000, E1    -6.546, E3 +167813.165}
SPL {X  -165.650, Y  +389.276, Z    +0.000, E1   -15.245, E3 +167812.673}
SPL {X  -165.650, Y  +395.801, Z    +0.000, E1   -28.236, E3 +167812.301}
SPL {X  -165.650, Y  +403.802, Z    +0.000, E1   -41.748, E3 +167812.121}
SPL {X  -165.650, Y  +419.045, Z    +0.000, E1   -60.641, E3 +167809.443}
SPL {X  -165.650, Y  +474.102, Z    +0.000, E1   -73.446, E3 +167821.226}
SPL {X  -165.650, Y  +640.142, Z    +0.000, E1   -72.635, E3 +167906.510}
ENDSPLINE

SPLINE
SPL {X  -165.650, Y  +612.217, Z    +0.000, E1   -68.647, E3 +167922.436}
ENDSPLINE

SPLINE
SPL {X  -165.650, Y  +623.643, Z    +0.000, E1   -68.543, E3 +167932.532}
SPL {X  -165.650, Y  +635.985, Z    +0.000, E1   -68.274, E3 +167944.911}
SPL {X  -165.650, Y  +656.072, Z    +0.000, E1   -68.403, E3 +167960.205}
SPL {X  -165.650, Y  +673.246, Z    +0.000, E1   -68.189, E3 +167975.961}
SPL {X  -164.760, Y  +692.647, Z    +0.000, E1   -68.400, E3 +167989.926}
SPL {X  -162.986, Y  +705.089, Z    +0.000, E1   -67.915, E3 +168004.138}
SPL {X  -159.812, Y  +719.091, Z    +0.000, E1   -67.711, E3 +168017.137}
SPL {X  -156.969, Y  +728.420, Z    +0.000, E1   -67.278, E3 +168027.919}
SPL {X  -154.751, Y  +734.593, Z    +0.000, E1   -66.864, E3 +168035.900}
SPL {X  -151.443, Y  +742.618, Z    +0.000, E1   -66.527, E3 +168044.895}
SPL {X  -146.969, Y  +751.920, Z    +0.000, E1   -66.066, E3 +168055.391}
SPL {X  -142.811, Y  +759.434, Z    +0.000, E1   -65.254, E3 +168066.240}
SPL {X  -139.420, Y  +764.954, Z    +0.000, E1   -64.577, E3 +168074.238}
SPL {X  -136.483, Y  +769.374, Z    +0.000, E1   -64.163, E3 +168079.893}
SPL {X  -133.523, Y  +773.539, Z    +0.000, E1   -63.962, E3 +168084.162}
SPL {X  -125.028, Y  +784.164, Z    +0.000, E1   -66.760, E3 +168080.237}
SPL {X   -71.589, Y  +824.882, Z    +0.000, E1   -56.415, E3 +168207.303}
ENDSPLINE

SPLINE
SPL {X  -127.072, Y  +781.767, Z    +0.000, E1   -54.186, E3 +168370.275}
SPL {X  -150.680, Y  +744.314, Z    +0.000, E1   -44.608, E3 +168381.231}
SPL {X  -162.376, Y  +708.273, Z    +0.000, E1   -25.870, E3 +168373.355}
SPL {X  -165.092, Y  +689.091, Z    +0.000, E1   -12.938, E3 +168374.773}
SPL {X  -165.569, Y  +680.695, Z    +0.000, E1    -6.245, E3 +168373.459}
SPL {X  -165.650, Y  +673.489, Z    +0.000, E1    -0.162, E3 +168372.963}
SPL {X  -165.650, Y  +669.039, Z    +0.000, E1    +7.218, E3 +168372.224}
SPL {X  -165.650, Y  +663.739, Z    +0.000, E1   +17.756, E3 +168371.915}
SPL {X  -165.650, Y  +656.188, Z    +0.000, E1   +32.567, E3 +168371.197}
SPL {X  -165.650, Y  +648.712, Z    +0.000, E1   +45.195, E3 +168370.819}
SPL {X  -165.650, Y  +636.657, Z    +0.000, E1   +60.410, E3 +168368.097}
SPL {X  -165.650, Y  +613.310, Z    +0.000, E1   +72.038, E3 +168368.456}
SPL {X  -165.650, Y  +568.914, Z    +0.000, E1   +74.438, E3 +168383.041}
SPL {X  -165.650, Y  +420.321, Z    +0.000, E1   +71.570, E3 +168471.694}
ENDSPLINE

SPLINE
SPL {X  -165.650, Y  +437.633, Z    +0.000, E1   +68.421, E3 +168487.443}
ENDSPLINE

SPLINE
SPL {X  -164.513, Y  +359.128, Z    +0.000, E1   +73.170, E3 +168497.676}
SPL {X  -163.967, Y  +354.944, Z    +0.000, E1   +72.327, E3 +168509.030}
SPL {X  -163.372, Y  +351.124, Z    +0.000, E1   +71.295, E3 +168521.622}
SPL {X  -162.653, Y  +347.134, Z    +0.000, E1   +70.371, E3 +168532.857}
SPL {X  -161.430, Y  +341.349, Z    +0.000, E1   +69.492, E3 +168544.932}
SPL {X  -160.389, Y  +337.084, Z    +0.000, E1   +68.301, E3 +168558.019}
SPL {X  -159.245, Y  +332.881, Z    +0.000, E1   +67.496, E3 +168567.679}
SPL {X  -157.072, Y  +325.885, Z    +0.000, E1   +67.020, E3 +168577.028}
SPL {X  -154.432, Y  +318.577, Z    +0.000, E1   +66.843, E3 +168584.233}
SPL {X  -151.047, Y  +310.495, Z    +0.000, E1   +66.593, E3 +168592.645}
SPL {X  -146.639, Y  +301.448, Z    +0.000, E1   +65.839, E3 +168604.854}
SPL {X  -142.469, Y  +293.987, Z    +0.000, E1   +65.133, E3 +168614.903}
SPL {X  -139.022, Y  +288.429, Z    +0.000, E1   +64.807, E3 +168621.101}
SPL {X  -136.717, Y  +284.968, Z    +0.000, E1   +64.044, E3 +168627.694}
SPL {X  -133.061, Y  +279.835, Z    +0.000, E1   +64.204, E3 +168631.107}
SPL {X  -118.927, Y  +263.191, Z    +0.000, E1   +67.951, E3 +168627.120}
SPL {X   -76.819, Y  +231.739, Z    +0.000, E1   +54.834, E3 +168805.126}
ENDSPLINE

SPLINE
SPL {X  -140.879, Y  +291.363, Z    +0.000, E1   +48.273, E3 +168912.567}
SPL {X  -158.845, Y  +331.507, Z    +0.000, E1   +33.834, E3 +168921.902}
SPL {X  -164.164, Y  +356.358, Z    +0.000, E1   +18.707, E3 +168918.224}
SPL {X  -165.341, Y  +368.384, Z    +0.000, E1   +10.076, E3 +168918.968}
SPL {X  -165.648, Y  +377.641, Z    +0.000, E1    +2.653, E3 +168918.319}
SPL {X  -165.650, Y  +380.500, Z    +0.000, E1    -0.000, E3 +168917.350}
SPL {X  -165.650, Y  +381.694, Z    +0.000, E1    -1.679, E3 +168916.751}
SPL {X  -165.650, Y  +384.595, Z    +0.000, E1    -6.546, E3 +168916.613}
SPL {X  -165.650, Y  +389.276, Z    +0.000, E1   -15.245, E3 +168916.122}
SPL {X  -165.650, Y  +395.801, Z    +0.000, E1   -28.236, E3 +168915.749}
SPL {X  -165.650, Y  +403.802, Z    +0.000, E1   -41.748, E3 +168915.570}
SPL {X  -165.650, Y  +419.045, Z    +0.000, E1   -60.641, E3 +168912.891}
SPL {X  -165.650, Y  +474.102, Z    +0.000, E1   -73.446, E3 +168924.674}
SPL {X  -165.650, Y  +640.142, Z    +0.000, E1   -72.635, E3 +169009.959}
ENDSPLINE

SPLINE
SPL {X  -165.650, Y  +612.217, Z    +0.000, E1   -68.647, E3 +169025.884}
ENDSPLINE

SPLINE
SPL {X  -165.650, Y  +623.643, Z    +0.000, E1   -68.543, E3 +169035.981}
SPL {X  -165.650, Y  +635.985, Z    +0.000, E1   -68.274, E3 +169048.359}
SPL {X  -165.650, Y  +656.072, Z    +0.000, E1   -68.403, E3 +169063.654}
SPL {X  -165.650, Y  +673.246, Z    +0.000, E1   -68.189, E3 +169079.409}
SPL {X  -164.760, Y  +692.647, Z    +0.000, E1   -68.400, E3 +169093.374}
SPL {X  -163.763, Y  +700.430, Z    +0.000, E1   -67.939, E3 +169103.397}
SPL {X  -161.478, Y  +712.444, Z    +0.000, E1   -67.895, E3 +169113.752}
SPL {X  -157.774, Y  +725.970, Z    +0.000, E1   -67.383, E3 +169128.754}
SPL {X  -153.458, Y  +737.875, Z    +0.000, E1   -66.902, E3 +169141.829}
SPL {X  -149.433, Y  +746.982, Z    +0.000, E1   -66.131, E3 +169154.460}
SPL {X  -144.642, Y  +756.238, Z    +0.000, E1   -65.678, E3 +169164.690}
SPL {X  -141.719, Y  +761.265, Z    +0.000, E1   -65.117, E3 +169171.823}
SPL {X  -139.420, Y  +764.954, Z    +0.000, E1   -64.577, E3 +169177.687}
SPL {X  -136.483, Y  +769.374, Z    +0.000, E1   -64.163, E3 +169183.342}
SPL {X  -133.523, Y  +773.539, Z    +0.000, E1   -63.962, E3 +169187.610}
SPL {X  -125.028, Y  +784.164, Z    +0.000, E1   -66.760, E3 +169183.686}
SPL {X   -71.589, Y  +824.882, Z    +0.000, E1   -56.415, E3 +169310.751}
ENDSPLINE

SPLINE
SPL {X  -127.072, Y  +781.767, Z    +0.000, E1   -54.186, E3 +169473.723}
SPL {X  -150.680, Y  +744.314, Z    +0.000, E1   -44.608, E3 +169484.679}
SPL {X  -162.376, Y  +708.273, Z    +0.000, E1   -25.870, E3 +169476.803}
SPL {X  -165.092, Y  +689.091, Z    +0.000, E1   -12.938, E3 +169478.222}
SPL {X  -165.629, Y  +678.122, Z    +0.000, E1    -4.178, E3 +169477.369}
SPL {X  -165.650, Y  +673.539, Z    +0.000, E1    -0.057, E3 +169476.466}
SPL {X  -165.650, Y  +671.359, Z    +0.000, E1    +3.116, E3 +169475.823}
SPL {X  -165.650, Y  +667.465, Z    +0.000, E1   +10.413, E3 +169475.618}
SPL {X  -165.650, Y  +662.220, Z    +0.000, E1   +20.600, E3 +169475.310}
SPL {X  -165.650, Y  +652.464, Z    +0.000, E1   +39.379, E3 +169474.257}
SPL {X  -165.650, Y  +636.657, Z    +0.000, E1   +60.410, E3 +169471.545}
SPL {X  -165.650, Y  +613.310, Z    +0.000, E1   +72.038, E3 +169471.905}
SPL {X  -165.650, Y  +568.914, Z    +0.000, E1   +74.438, E3 +169486.489}
SPL {X  -165.650, Y  +420.321, Z    +0.000, E1   +71.570, E3 +169575.143}
ENDSPLINE

SPLINE
SPL {X  -165.650, Y  +437.633, Z    +0.000, E1   +68.421, E3 +169590.891}
ENDSPLINE

SPLINE
SPL {X  -164.513, Y  +359.128, Z    +0.000, E1   +73.170, E3 +169601.125}
SPL {X  -163.967, Y  +354.944, Z    +0.000, E1   +72.327, E3 +169612.478}
SPL {X  -163.372, Y  +351.124, Z    +0.000, E1   +71.295, E3 +169625.070}
SPL {X  -162.653, Y  +347.134, Z    +0.000, E1   +70.371, E3 +169636.306}
SPL {X  -161.430, Y  +341.349, Z    +0.000, E1   +69.492, E3 +169648.380}
SPL {X  -160.389, Y  +337.084, Z    +0.000, E1   +68.301, E3 +169661.467}
SPL {X  -159.245, Y  +332.881, Z    +0.000, E1   +67.496, E3 +169671.127}
SPL {X  -157.072, Y  +325.885, Z    +0.000, E1   +67.020, E3 +169680.476}
SPL {X  -154.432, Y  +318.577, Z    +0.000, E1   +66.843, E3 +169687.681}
SPL {X  -151.047, Y  +310.495, Z    +0.000, E1   +66.593, E3 +169696.093}
SPL {X  -146.639, Y  +301.448, Z    +0.000, E1   +65.839, E3 +169708.302}
SPL {X  -142.469, Y  +293.987, Z    +0.000, E1   +65.133, E3 +169718.351}
SPL {X  -139.022, Y  +288.429, Z    +0.000, E1   +64.807, E3 +169724.549}
SPL {X  -136.717, Y  +284.968, Z    +0.000, E1   +64.044, E3 +169731.142}
SPL {X  -133.061, Y  +279.835, Z    +0.000, E1   +64.204, E3 +169734.555}
SPL {X  -118.927, Y  +263.191, Z    +0.000, E1   +67.951, E3 +169730.568}
SPL {X   -76.819, Y  +231.739, Z    +0.000, E1   +54.834, E3 +169908.574}
ENDSPLINE

SPLINE
SPL {X  -140.879, Y  +291.363, Z    +0.000, E1   +48.273, E3 +170016.015}
SPL {X  -158.845, Y  +331.507, Z    +0.000, E1   +33.834, E3 +170025.350}
SPL {X  -164.164, Y  +356.358, Z    +0.000, E1   +18.707, E3 +170021.672}
SPL {X  -165.341, Y  +368.384, Z    +0.000, E1   +10.076, E3 +170022.417}
SPL {X  -165.648, Y  +377.641, Z    +0.000, E1    +2.653, E3 +170021.767}
SPL {X  -165.650, Y  +380.500, Z    +0.000, E1    -0.000, E3 +170020.798}
SPL {X  -165.650, Y  +381.694, Z    +0.000, E1    -1.679, E3 +170020.200}
SPL {X  -165.650, Y  +384.595, Z    +0.000, E1    -6.546, E3 +170020.062}
SPL {X  -165.650, Y  +389.276, Z    +0.000, E1   -15.245, E3 +170019.570}
SPL {X  -165.650, Y  +395.801, Z    +0.000, E1   -28.236, E3 +170019.197}
SPL {X  -165.650, Y  +403.802, Z    +0.000, E1   -41.748, E3 +170019.018}
SPL {X  -165.650, Y  +419.045, Z    +0.000, E1   -60.641, E3 +170016.339}
SPL {X  -165.650, Y  +474.102, Z    +0.000, E1   -73.446, E3 +170028.122}
SPL {X  -165.650, Y  +640.142, Z    +0.000, E1   -72.635, E3 +170113.407}
ENDSPLINE

SPLINE
SPL {X  -165.650, Y  +612.217, Z    +0.000, E1   -68.647, E3 +170129.332}
ENDSPLINE

SPLINE
SPL {X  -165.650, Y  +623.643, Z    +0.000, E1   -68.543, E3 +170139.429}
SPL {X  -165.650, Y  +635.985, Z    +0.000, E1   -68.274, E3 +170151.807}
SPL {X  -165.650, Y  +656.072, Z    +0.000, E1   -68.403, E3 +170167.102}
SPL {X  -165.650, Y  +673.246, Z    +0.000, E1   -68.189, E3 +170182.857}
SPL {X  -164.760, Y  +692.647, Z    +0.000, E1   -68.400, E3 +170196.822}
SPL {X  -162.986, Y  +705.089, Z    +0.000, E1   -67.915, E3 +170211.034}
SPL {X  -159.812, Y  +719.091, Z    +0.000, E1   -67.711, E3 +170224.033}
SPL {X  -156.969, Y  +728.420, Z    +0.000, E1   -67.278, E3 +170234.815}
SPL {X  -153.458, Y  +737.875, Z    +0.000, E1   -66.902, E3 +170245.277}
SPL {X  -149.433, Y  +746.982, Z    +0.000, E1   -66.131, E3 +170257.908}
SPL {X  -144.642, Y  +756.238, Z    +0.000, E1   -65.678, E3 +170268.139}
SPL {X  -140.398, Y  +763.411, Z    +0.000, E1   -64.853, E3 +170278.615}
SPL {X  -135.180, Y  +771.240, Z    +0.000, E1   -64.104, E3 +170288.664}
SPL {X  -125.028, Y  +784.164, Z    +0.000, E1   -66.760, E3 +170287.134}
SPL {X   -71.589, Y  +824.882, Z    +0.000, E1   -56.415, E3 +170414.199}
ENDSPLINE

SPLINE
SPL {X  -127.072, Y  +781.767, Z    +0.000, E1   -54.186, E3 +170577.171}
SPL {X  -150.680, Y  +744.314, Z    +0.000, E1   -44.608, E3 +170588.127}
SPL {X  -162.376, Y  +708.273, Z    +0.000, E1   -25.870, E3 +170580.251}
SPL {X  -165.092, Y  +689.091, Z    +0.000, E1   -12.938, E3 +170581.670}
SPL {X  -165.629, Y  +678.122, Z    +0.000, E1    -4.178, E3 +170580.817}
SPL {X  -165.650, Y  +673.539, Z    +0.000, E1    -0.057, E3 +170579.915}
SPL {X  -165.650, Y  +671.359, Z    +0.000, E1    +3.116, E3 +170579.272}
SPL {X  -165.650, Y  +665.277, Z    +0.000, E1   +14.409, E3 +170578.916}
SPL {X  -165.650, Y  +659.573, Z    +0.000, E1   +26.182, E3 +170578.664}
SPL {X  -165.650, Y  +652.464, Z    +0.000, E1   +39.379, E3 +170577.705}
SPL {X  -165.650, Y  +634.871, Z    +0.000, E1   +61.762, E3 +170574.938}
SPL {X  -165.650, Y  +574.769, Z    +0.000, E1   +74.441, E3 +170587.586}
SPL {X  -165.650, Y  +420.321, Z    +0.000, E1   +71.570, E3 +170678.591}
ENDSPLINE

SPLINE
SPL {X  -165.650, Y  +437.633, Z    +0.000, E1   +68.421, E3 +170694.339}
ENDSPLINE

SPLINE
SPL {X  -164.513, Y  +359.128, Z    +0.000, E1   +73.170, E3 +170704.573}
SPL {X  -163.967, Y  +354.944, Z    +0.000, E1   +72.327, E3 +170715.926}
SPL {X  -163.372, Y  +351.124, Z    +0.000, E1   +71.295, E3 +170728.518}
SPL {X  -162.653, Y  +347.134, Z    +0.000, E1   +70.371, E3 +170739.754}
SPL {X  -161.430, Y  +341.349, Z    +0.000, E1   +69.492, E3 +170751.828}
SPL {X  -160.389, Y  +337.084, Z    +0.000, E1   +68.301, E3 +170764.915}
SPL {X  -158.795, Y  +331.340, Z    +0.000, E1   +67.291, E3 +170777.602}
SPL {X  -155.058, Y  +320.218, Z    +0.000, E1   +66.982, E3 +170788.908}
SPL {X  -151.047, Y  +310.495, Z    +0.000, E1   +66.593, E3 +170799.541}
SPL {X  -148.187, Y  +304.469, Z    +0.000, E1   +66.029, E3 +170807.920}
SPL {X  -145.703, Y  +299.692, Z    +0.000, E1   +65.663, E3 +170814.087}
SPL {X  -142.469, Y  +293.987, Z    +0.000, E1   +65.133, E3 +170821.799}
SPL {X  -139.022, Y  +288.429, Z    +0.000, E1   +64.807, E3 +170827.998}
SPL {X  -136.717, Y  +284.968, Z    +0.000, E1   +64.044, E3 +170834.590}
SPL {X  -133.061, Y  +279.835, Z    +0.000, E1   +64.204, E3 +170838.004}
SPL {X  -118.927, Y  +263.191, Z    +0.000, E1   +67.951, E3 +170834.016}
SPL {X   -75.220, Y  +230.913, Z    +0.000, E1   +55.539, E3 +170974.648}
ENDSPLINE

SPLINE
SPL {X   -78.274, Y  +232.510, Z    +0.000, E1   +54.798, E3 +171025.130}
SPL {X  -140.879, Y  +291.363, Z    +0.000, E1   +48.273, E3 +171119.463}
SPL {X  -155.054, Y  +320.205, Z    +0.000, E1   +39.591, E3 +171131.915}
SPL {X  -160.978, Y  +339.437, Z    +0.000, E1   +29.257, E3 +171126.545}
SPL {X  -164.164, Y  +356.358, Z    +0.000, E1   +18.707, E3 +171125.121}
SPL {X  -165.519, Y  +371.910, Z    +0.000, E1    +7.409, E3 +171125.530}
SPL {X  -165.650, Y  +380.329, Z    +0.000, E1    +0.239, E3 +171124.376}
SPL {X  -165.650, Y  +381.694, Z    +0.000, E1    -1.679, E3 +171123.648}
SPL {X  -165.650, Y  +384.595, Z    +0.000, E1    -6.546, E3 +171123.510}
SPL {X  -165.650, Y  +389.276, Z    +0.000, E1   -15.245, E3 +171123.018}
SPL {X  -165.650, Y  +395.801, Z    +0.000, E1   -28.236, E3 +171122.645}
SPL {X  -165.650, Y  +403.802, Z    +0.000, E1   -41.748, E3 +171122.466}
SPL {X  -165.650, Y  +419.045, Z    +0.000, E1   -60.641, E3 +171119.787}
SPL {X  -165.650, Y  +474.102, Z    +0.000, E1   -73.446, E3 +171131.571}
SPL {X  -165.650, Y  +640.142, Z    +0.000, E1   -72.635, E3 +171216.855}
ENDSPLINE

SPLINE
SPL {X  -165.650, Y  +619.423, Z    +0.000, E1   -68.618, E3 +171239.053}
ENDSPLINE

SPLINE
SPL {X  -165.650, Y  +635.985, Z    +0.000, E1   -68.274, E3 +171255.256}
SPL {X  -165.650, Y  +647.687, Z    +0.000, E1   -68.151, E3 +171265.756}
SPL {X  -165.650, Y  +665.917, Z    +0.000, E1   -68.414, E3 +171278.515}
SPL {X  -165.417, Y  +684.287, Z    +0.000, E1   -68.467, E3 +171292.812}
SPL {X  -164.268, Y  +696.853, Z    +0.000, E1   -68.071, E3 +171306.441}
SPL {X  -162.443, Y  +707.938, Z    +0.000, E1   -67.853, E3 +171317.176}
SPL {X  -159.812, Y  +719.091, Z    +0.000, E1   -67.711, E3 +171327.481}
SPL {X  -156.969, Y  +728.420, Z    +0.000, E1   -67.278, E3 +171338.264}
SPL {X  -154.751, Y  +734.593, Z    +0.000, E1   -66.864, E3 +171346.245}
SPL {X  -151.443, Y  +742.618, Z    +0.000, E1   -66.527, E3 +171355.239}
SPL {X  -146.969, Y  +751.920, Z    +0.000, E1   -66.066, E3 +171365.736}
SPL {X  -142.811, Y  +759.434, Z    +0.000, E1   -65.254, E3 +171376.585}
SPL {X  -139.420, Y  +764.954, Z    +0.000, E1   -64.577, E3 +171384.583}
SPL {X  -136.483, Y  +769.374, Z    +0.000, E1   -64.163, E3 +171390.238}
SPL {X  -133.523, Y  +773.539, Z    +0.000, E1   -63.962, E3 +171394.507}
SPL {X  -125.028, Y  +784.164, Z    +0.000, E1   -66.760, E3 +171390.582}
SPL {X   -71.589, Y  +824.882, Z    +0.000, E1   -56.415, E3 +171517.647}
ENDSPLINE

SPLINE
SPL {X  -127.072, Y  +781.767, Z    +0.000, E1   -54.186, E3 +171680.619}
SPL {X  -150.680, Y  +744.314, Z    +0.000, E1   -44.608, E3 +171691.576}
SPL {X  -162.376, Y  +708.273, Z    +0.000, E1   -25.870, E3 +171683.699}
SPL {X  -165.092, Y  +689.091, Z    +0.000, E1   -12.938, E3 +171685.118}
SPL {X  -165.629, Y  +678.122, Z    +0.000, E1    -4.178, E3 +171684.265}
SPL {X  -165.650, Y  +673.539, Z    +0.000, E1    -0.057, E3 +171683.363}
SPL {X  -165.650, Y  +671.359, Z    +0.000, E1    +3.116, E3 +171682.720}
SPL {X  -165.650, Y  +665.277, Z    +0.000, E1   +14.409, E3 +171682.365}
SPL {X  -165.650, Y  +659.573, Z    +0.000, E1   +26.182, E3 +171682.113}
SPL {X  -165.650, Y  +652.464, Z    +0.000, E1   +39.379, E3 +171681.154}
SPL {X  -165.650, Y  +634.871, Z    +0.000, E1   +61.762, E3 +171678.386}
SPL {X  -165.650, Y  +574.769, Z    +0.000, E1   +74.441, E3 +171691.034}
SPL {X  -165.650, Y  +420.321, Z    +0.000, E1   +71.570, E3 +171782.039}
ENDSPLINE

SPLINE
SPL {X  -165.650, Y  +437.633, Z    +0.000, E1   +68.421, E3 +171797.788}
ENDSPLINE

SPLINE
SPL {X  -164.513, Y  +359.128, Z    +0.000, E1   +73.170, E3 +171808.021}
SPL {X  -163.967, Y  +354.944, Z    +0.000, E1   +72.327, E3 +171819.375}
SPL {X  -163.372, Y  +351.124, Z    +0.000, E1   +71.295, E3 +171831.967}
SPL {X  -162.653, Y  +347.134, Z    +0.000, E1   +70.371, E3 +171843.202}
SPL {X  -161.451, Y  +341.438, Z    +0.000, E1   +69.889, E3 +171851.521}
SPL {X  -161.195, Y  +340.340, Z    +0.000, E1   +68.690, E3 +171862.742}
SPL {X  -159.328, Y  +333.173, Z    +0.000, E1   +67.752, E3 +171875.963}
SPL {X  -157.072, Y  +325.885, Z    +0.000, E1   +67.020, E3 +171887.373}
SPL {X  -153.570, Y  +316.402, Z    +0.000, E1   +66.799, E3 +171896.734}
SPL {X  -149.308, Y  +306.758, Z    +0.000, E1   +66.321, E3 +171907.860}
SPL {X  -145.703, Y  +299.692, Z    +0.000, E1   +65.663, E3 +171917.535}
SPL {X  -142.469, Y  +293.987, Z    +0.000, E1   +65.133, E3 +171925.247}
SPL {X  -139.022, Y  +288.429, Z    +0.000, E1   +64.807, E3 +171931.446}
SPL {X  -136.717, Y  +284.968, Z    +0.000, E1   +64.044, E3 +171938.038}
SPL {X  -133.061, Y  +279.835, Z    +0.000, E1   +64.204, E3 +171941.452}
SPL {X  -118.927, Y  +263.191, Z    +0.000, E1   +67.951, E3 +171937.464}
SPL {X   -76.819, Y  +231.739, Z    +0.000, E1   +54.834, E3 +172115.471}
ENDSPLINE

